(* CODESYS project CtaAppBacNetKBOB_1.0.0.0.library
   Description: CtaAppBacNetKBOB Library der CTA
   Version: 1.0.0.0
   Title: CtaAppBacNetKBOB
   Author: SIS
   Company: CTA
   DocFormat: reStructuredText
   Placeholder: CtaAppBacNetKBOB
   DefaultNamespace: CtaAppBacNetKBOB
   CompiledLibraryCompatibilityVersion: CODESYS V3.5 SP16 Patch 3
   LanguageModelAttribute: qualified-access-only

Project tree, tasks and I/O mapping:
  libraries: CtaAppBmk, 1.0.0.0 (CTA); Standard, 3.5.18.0 (System); CtaSysConfig, 1.0.0.0 (CTA); CmpDynamicText, 3.5.17.0 (System); WagoTypesBACnet, 1.0.9.7 (WAGO); SysProcess, 3.5.17.0 (System); CtaVisSymbols, 1.0.0.0 (CTA); StringUtils, 3.5.18.0 (System); SysTypes2 Interfaces, * (System); VisuSymbols, 4.5.0.0 (System); CtaVisHelp, 1.0.0.0 (CTA); WagoSysErrorBase, 1.6.2.6 (WAGO); WagoSysBACnet, 2.0.0.6 (WAGO); WagoSysVisuBACnet, 2.0.0.0 (WAGO)
  40 Visualizations/
    BACNET_PARAMETER/
      visualisation DIA_BACNET_PARAMETER
      visualisation VIS_DIA_BACNET_PARAMETER
      visualisation VIS_BACNET_APP
      visualisation DIA_BACNET_LIST
  30 Program Organization Units/
    FCs/
      XMLFcs/
        XMLBase/
          function fcXMLAddAttribute [ST]
          function fcXMLCheckNode [ST]
          function fcXMLDeleteNode [ST]
          function fcXMLUpdateAttribute [ST]
          function fcXMLUpdateNode [ST]
          function fcXMLAddNode [ST]
        XML BacNet Override/
          DELETENODE/
            function fcXMLDeleteOverrideNode [ST]
          STRUCTUREDVIEW/
            function fcXMLStructuredView [ST]
            function fcXMLAddStructuredViewToDevice [ST]
            function fcXMLDeleteStructuredViewFromDevice [ST]
          TRENDLOG/
            function fcXMLTrendLogOverride [ST]
          DEVICE/
            function fcXMLDeviceOverride [ST]
      BacNetId/
        function fcDWordToHexString [ST]
        function fcBacNetIdToIdWitType [ST]
      BmkToAdr/
        function fcBmkToAdr [ST]
      BacNetText/
        function fcGetBcText [ST]
      UTF8Fcs/
        function fcAsciiToUtf [ST]
        function fcUtfToAscii [ST]
      BacNetIni/
        function fcBacNetIni [ST]
    FBs/
      AT_FUNKTIONEN/
        AT_MESSWERTGEBER_BINÄR/
          function block FB_AT_MESSWERTGEBER_BINÄR [ST]: metDELETE, metCREATE, metCreate_A_BI_1, metCreate_B_TL_1, metCreate_C_BV_1, metCREATE_KBOB_2017_V1, metCREATE_STRUCTVIEW_KBOB_2017_V1, metCREATE_STRUCTVIEW_KBOB_2021_V2, metCREATE_KBOB_2021_V2, FB_EXIT, metCYCLIC_DESCRIPTION_FIX, metCYCLIC_KBOB_2017_V1, metCYCLIC_KBOB_2021_V2
        AT_MESSWERTGEBER_STETIG/
          function block FB_AT_MESSWERTGEBER_STETIG [ST]: metDELETE, FB_EXIT, metCREATE, metCreate_A_AI_1, metCreate_C_TL_1, metCreate_B_EE_1, metCREATE_KBOB_2017_V1, metCREATE_STRUCTVIEW_KBOB_2017_V1, metCREATE_KBOB_2021_V2, metCREATE_STRUCTVIEW_KBOB_2021_V2, metCYCLIC_KBOB_2017_V1, metCYCLIC_KBOB_2021_V2, metCYCLIC_DESCRIPTION_FIX
        AT_ANTRIEB_STETIG/
          function block FB_AT_ANTRIEB_STETIG [ST]: metCYCLIC_KBOB_2017_V1, metCYCLIC_KBOB_2021_V2, metCYCLIC_DESCRIPTION_FIX, FB_EXIT, metDELETE, metCREATE_KBOB_2017_V1, metCREATE_STRUCTVIEW_KBOB_2017_V1, metCREATE_STRUCTVIEW_KBOB_2021_V2, metCREATE_KBOB_2021_V2, metCREATE, metCreate_F_BI_1, metCreate_G_AO_1, metCreate_I_AI_1, metCreate_K_BI_2, metCreate_L_BV_3, metCreate_H_TL_2, metCreate_J_TL_3, metCreate_A_BO_1, metCreate_B_TL_1, metCreate_C_EE_1, metCreate_E_BV_2
        AT_ANLAGENSCHALTER/
          function block FB_AT_ANLAGENSCHALTER [ST]: FB_EXIT, metCREATE, metCreate_A_MV_1, metCreate_B_MI_1, metCreate_C_BV_1, metCreate_D_SC_1, metCREATE_KBOB_2017_V1, metCREATE_STRUCTVIEW_KBOB_2017_V1, metCREATE_KBOB_2021_V2, metCREATE_STRUCTVIEW_KBOB_2021_V2, metDELETE, metCYCLIC_KBOB_2017_V1, metCYCLIC_KBOB_2021_V2, metCYCLIC_DESCRIPTION_FIX
        AT_AUTOMATIONSTATION/
          function block FB_AT_AUTOMATIONSSTATION [ST]: metCYCLIC_KBOB_2017_V1, metCYCLIC_KBOB_2021_V2, metCYCLIC_DESCRIPTION_FIX, FB_EXIT, metDELETE, metCREATE_KBOB_2017_V1, metCREATE_STRUCTVIEW_KBOB_2017_V1, metCREATE_KBOB_2021_V2, metCREATE_STRUCTVIEW_KBOB_2021_V2, metCREATE, metCreate_L_NC_160, metCreate_L_NC_161, metCreate_L_NC_162, metCreate_L_NC_163, metCreate_M_NC_192, metCreate_M_NC_193, metCreate_N_NC_224, metCreate_N_NC_225, metCreate_O_BV_1, metCreate_P_BV_2, metCreate_Q_BV_3, metCreate_R_BV_4, metCreate_S_BV_5, metCreate_I_NC_66, metCreate_J_NC_97, metCreate_J_NC_98, metCreate_J_NC_99, metCreate_K_NC_128, metCreate_H_NC_35, metCreate_I_NC_64, metCreate_I_NC_67, metCreate_J_NC_96, metCreate_K_NC_129, metCreate_K_NC_130, metCreate_K_NC_131, metCreate_A_DV_1, metCreate_B_CL_1, metCreate_C_CL_2, metCreate_D_CL_3, metCreate_E_CL_4, metCreate_F_EL_1, metCreate_G_NC_1, metCreate_G_NC_2, metCreate_G_NC_3, metCreate_G_NC_4, metCreate_H_NC_32, metCreate_H_NC_33, metCreate_H_NC_34, metCreate_I_NC_65
        AT_ANLAGEFUNKTION/
          function block FB_AT_ANLAGEFUNKTION [ST]: metCREATE_STRUCTVIEW_KBOB_2021_V2, metCREATE_KBOB_2021_V2, metCreate_H_BO_2, metCreate_I_BO_3, metCreate_D_BV_4, metCreate_E_BI_1, metCreate_B_BV_2, metCreate_C_BV_3, metCreate_J_SC_1, metCreate_F_BV_5, metCreate_G_BO_1, metCreate_A_BV_1, metCREATE_KBOB_2017_V1, metCREATE_STRUCTVIEW_KBOB_2017_V1, metCREATE, metCYCLIC_KBOB_2017_V1, metCYCLIC_KBOB_2021_V2, metCYCLIC_DESCRIPTION_FIX, FB_EXIT, metDELETE
        AT_ZÄHLER/
          function block FB_AT_ZÄHLER [ST]: metCREATE_STRUCTVIEW_KBOB_2021_V2, metCREATE_KBOB_2021_V2, metCreate_A_AV_1, metCreate_B_TL_1, metCreate_C_BV_1, metCREATE, metCREATE_KBOB_2017_V1, metCREATE_STRUCTVIEW_KBOB_2017_V1, metDELETE, FB_EXIT, metCYCLIC_DESCRIPTION_FIX, metCYCLIC_KBOB_2017_V1, metCYCLIC_KBOB_2021_V2
        AT_STELLORGAN_STETIG/
          function block FB_AT_AT_STELLORGAN_STETIG [ST]: metCREATE_STRUCTVIEW_KBOB_2021_V2, metCREATE_KBOB_2021_V2, metCreate_D_BI_1, metCreate_A_AO_1, metCreate_C_TL_1, metCreate_E_BI_2, metCreate_B_AI_1, metCreate_F_BV_1, metCREATE_KBOB_2017_V1, metCREATE_STRUCTVIEW_KBOB_2017_V1, metCREATE, metCYCLIC_KBOB_2017_V1, metCYCLIC_KBOB_2021_V2, metCYCLIC_DESCRIPTION_FIX, FB_EXIT, metDELETE
      BACNET_PARAMETER/
        function block FB_BACNET_PARAMETER [ST]: proCreate, proDelete, proUseAKS, proInitDone, CONFIG, metRequestDelete, metGetTextListName, proKBOB_REV, P_fbenBacNetKbobRev, P_fbxEnableBacNet, P_fbxUseAKS, P_fbxUseExklTxtList, proTimeToOnline, proDestroyBacNetOverrideXmlNode, proRebootRequired, metAddObj, BACNETLIBPARACHECK, P_fbdiDeviceId, P_fbxAnsiCodiert
      OBJ_IDENTIFER_BASE/
        function block FB_OBJ_ID_BASE [ST]: OBJ_ID_BASE, OBJ_NAME_BASE, OBJ_NAME_DESCRIPTION, metCREATE, metDELETE, FB_EXIT, FB_INIT, proINextObj, proIsCreatet, proAllowCreate, proAllowDelete
    Pou/
      program BAC_NET [ST]
  00000000-0000-0000-0000-000000000000|D:\CoDeSys\LibrariesV3\trunk\Intern\CAA\CAA Template\3.4.0.0 draft\Placeholder.xml
  00000000-0000-0000-0000-000000000000|D:\CoDeSys\LibrariesV3\trunk\Intern\CAA\CAA Template\3.2.0.3 draft\Prefix.pdf
  00000000-0000-0000-0000-000000000000|D:\CoDeSys\LibrariesV3\trunk\Intern\CAA\CAA Template\3.5.2.0 draft\Placeholder.xml
  20 Structs/
    ENUMERATION/
      data type enTypeOfBacNetFunktion
      data type enEvent
      data type enTypeOfBacNetTextList
      data type enKBOB_REV
  50 Images/
  10 Documenation/
    global variables VersionHistory
    global variables readMe
  21 Interface/
    BACNET_PARAMETER/
      interface ITF_BACNET_PARAMETER: metGetTextListName, metRequestDelete, proCreate, proDelete, proInitDone, proKBOB_REV, proUseAKS, P_fbxEnableBacNet, P_fbxUseAKS, P_fbxUseExklTxtList, P_fbenBacNetKbobRev, proTimeToOnline, metAddObj, proRebootRequired, proDestroyBacNetOverrideXmlNode, P_fbdiDeviceId, P_fbxAnsiCodiert
    OBJ_IDENTIFER_BASE/
      interface ITF_OBJ_ID_BASE: FB_EXIT, metCREATE, OBJ_ID_BASE, OBJ_NAME_BASE, OBJ_NAME_DESCRIPTION, metDELETE, proINextObj, proAllowCreate, proIsCreatet, proAllowDelete
  11 Library Parameter/
  12 Konstanten/
  60 Textlisten/
    AT_FUNKTIONEN_TEXTLISTEN/
      AT_ANLAGENSCHALTER/
        text list TXT_AT_ANLAGENSCHALTER_NC
        text list TXT_AT_ANLAGENSCHALTER_ENDING
        text list TXT_AT_ANLAGENSCHALTER_EVENTMESSAGE
        text list TXT_AT_ANLAGENSCHALTER_PRESV
        text list TXT_AT_ANLAGENSCHALTER_DESCRIPTION
      AT_ANTRIEB_STETIG/
        text list TXT_AT_ANTRIEB_STETIG_ENDING
        text list TXT_AT_ANTRIEB_STETIG_DESCRIPTION
        text list TXT_AT_ANTRIEB_STETIG_PRESV
        text list TXT_AT_ANTRIEB_STETIG_EVENTMESSAGE
        text list TXT_AT_ANTRIEB_STETIG_NC
      AT_MESSWERTGEBER_BINÄR/
        text list TXT_AT_MESSWERTGEBER_BINAR_DESCRIPTION
        text list TXT_AT_MESSWERTGEBER_BINAR_ENDING
        text list TXT_AT_MESSWERTGEBER_BINAR_NC
        text list TXT_AT_MESSWERTGEBER_BINAR_EVENTMESSAGE
        text list TXT_AT_MESSWERTGEBER_BINAR_PRESV
      AT_MESSWERTGEBER_STETIG/
        text list TXT_AT_MESSWERTGEBER_STETIG_NC
        text list TXT_AT_MESSWERTGEBER_STETIG_DESCRIPTION
        text list TXT_AT_MESSWERTGEBER_STETIG_ENDING
        text list TXT_AT_MESSWERTGEBER_STETIG_EVENTMESSAGE
        text list TXT_AT_MESSWERTGEBER_STETIG_PRESV
      AT_AUTOMATIONSTATION/
        text list TXT_AT_AUTOMATIONSSTATION_DESCRIPTION
        text list TXT_AT_AUTOMATIONSSTATION_ENDING
        text list TXT_AT_AUTOMATIONSSTATION_NC
        text list TXT_AT_AUTOMATIONSSTATION_PRESV
        text list TXT_AT_AUTOMATIONSSTATION_EVENTMESSAGE
      AT_ANLAGEFUNKTION/
        text list TXT_AT_ANLAGEFUNKTION_DESCRIPTION
        text list TXT_AT_ANLAGEFUNKTION_ENDING
        text list TXT_AT_ANLAGEFUNKTION_EVENTMESSAGE
        text list TXT_AT_ANLAGEFUNKTION_NC
        text list TXT_AT_ANLAGEFUNKTION_PRESV
      AT_ZÄHLER/
        text list TXT_AT_ZÄHLER_DESCRIPTION
        text list TXT_AT_ZÄHLER_ENDING
        text list TXT_AT_ZÄHLER_EVENTMESSAGE
        text list TXT_AT_ZÄHLER_NC
        text list TXT_AT_ZÄHLER_PRESV
      AT_STELLORGAN_STETIG/
        text list TXT_AT_STELLORGAN_STETIG_ENDING
        text list TXT_AT_STELLORGAN_STETIG_EVENTMESSAGE
        text list TXT_AT_STELLORGAN_STETIG_DESCRIPTION
        text list TXT_AT_STELLORGAN_STETIG_NC
        text list TXT_AT_STELLORGAN_STETIG_PRESV
    KBOB/
      text list KBOB_REV_TXT
  13 Globale Variablen/
    global variables GVL_BACNET
  text list GlobalTextList
*)

// 20 Structs/ENUMERATION/enTypeOfBacNetFunktion
{attribute 'qualified_only'}
TYPE enTypeOfBacNetFunktion :
(
	Type_Anlagenschalter            := 01,
    Type_AntriebStetig              := 02,
    Type_AbsperrStellorgan2p        := 03,
    Type_AbsperrStellorganStetig    := 04,
    Type_MesswertgeberStetig        := 05,
    Type_MesswertgeberBinär         := 06,
    Type_ParameterAnalog            := 07,
    Type_ParameterBinär             := 08,
	Type_Automationsstation			:= 09,
	Type_Anlagefunktion				:= 10,
	Type_Zähler						:= 11
);
END_TYPE

// 20 Structs/ENUMERATION/enEvent
{attribute 'qualified_only'}
{attribute 'strict'}
TYPE enEvent :
(
	ToOffNormal := 1,
	ToFault		:= 2,
	ToNormal	:= 3
);
END_TYPE

// 20 Structs/ENUMERATION/enTypeOfBacNetTextList
{attribute 'qualified_only'}
{attribute 'strict'}
TYPE enTypeOfBacNetTextList :
(
	ENDING 			:= 0,
	DESCRIPTION		:= 1,
	NC				:= 2,
	EVENTMESSAGE	:= 3,
	PRESENTVALUE	:= 4
);
END_TYPE

// 20 Structs/ENUMERATION/enKBOB_REV
{attribute 'qualified_only'}
TYPE enKBOB_REV :
(
	
	KBOB_REV2017_V1 := 0,
	KBOB_REV2021_V2 := 1
);
END_TYPE

// 10 Documenation/VersionHistory
(* 

.. image:: ../../Images/CTA_Logo.jpg
   :align: right
   :width: 15% 

**Vorlage**   


============ =========== =========== ============================================
**Date**     **Version** **Author**  **Change**
------------ ----------- ----------- --------------------------------------------
04.03.2021   0.0.0.0     SIS         Vorlage erstellt

============ =========== =========== ============================================


*)
VAR_GLOBAL
    stInfo : STRING:= '0.0.0.0, Vorlage, CTA';
END_VAR

// 10 Documenation/readMe
(*

**ReadMe**
 
|	**Empfehlung**
|
|	Dokumentrieren Sie die Library für eine nachhaltige Entwicklung
|     
| *Beispiel* 
|
| Dies ist die Vorlage Library der CTA. Erstellen Sie ihre Library anhand dieser Vorlage.
*)

VAR_GLOBAL
    xReadMeDone              :   BOOL;
END_VAR

// 13 Globale Variablen/GVL_BACNET
{attribute 'qualified_only'}
{attribute 'global_init_slot' := '49989'}
VAR_GLOBAL
	fbBacNetBmkDevice			:	CtaAppBmk.fbBMK := (stObjId := 'BacNetDevice');
	fbBacNetParameter			:	FB_BACNET_PARAMETER;
	fbAtAutomationsstation		:	FB_AT_AUTOMATIONSSTATION := (ITF_BMK_IN := fbBacNetBmkDevice);
	stBacNetDeviceId			:	STRING(8);
END_VAR

// 30 Program Organization Units/FCs/XMLFcs/XMLBase/fcXMLAddAttribute
FUNCTION fcXMLAddAttribute : BOOL
VAR_INPUT
	stParentPath			:	STRING(100);	// Start with '//*/
	stNodeName				:	STRING(100);
	stAttribute1			:	STRING(100);
	stAttribute1Value		:	STRING(150);
	stAttribute2Check		:	STRING(100);
	stAttribute2ValueCheck	:	STRING(150);
	stXmlFilePathName		:	STRING(255);
	xIgnoreCheck			:	BOOL;
END_VAR
VAR
	stCommand			:	STRING(1000);
	stTemp				:	STRING(255);
	stResult			:	STRING(255);
	RTS_IEC_RESULT		:	SysTypes.RTS_IEC_RESULT;
END_VAR

IF NOT fcXMLCheckNode(stParentPath,stNodeName,stAttribute1,stAttribute1Value,stAttribute2Check,stAttribute2ValueCheck,stXmlFilePathName) OR xIgnoreCheck THEN
	// create Attribute	
	stCommand := 	'';
	stTemp	  := 	'';
	stTemp	  :=	'xmlstarlet ed -L --insert "';
	StrConcatA(ADR(stTemp),ADR(stCommand),TO_INT(SIZEOF(stCommand)));
	stTemp	  := 	'';
	stTemp	  :=	stParentPath;
	StrConcatA(ADR(stTemp),ADR(stCommand),TO_INT(SIZEOF(stCommand)));
	stTemp	  := 	'';
	stTemp	  :=	'/';
	StrConcatA(ADR(stTemp),ADR(stCommand),TO_INT(SIZEOF(stCommand)));	
	stTemp	  := 	'';
	stTemp	  :=	stNodeName;
	StrConcatA(ADR(stTemp),ADR(stCommand),TO_INT(SIZEOF(stCommand)));	
	stTemp	  := 	'';
	stTemp	  :=	'[last()]" -t attr -n "';
	StrConcatA(ADR(stTemp),ADR(stCommand),TO_INT(SIZEOF(stCommand)));		
	stTemp	  := 	'';
	stTemp	  :=	stAttribute1;
	StrConcatA(ADR(stTemp),ADR(stCommand),TO_INT(SIZEOF(stCommand)));	
	stTemp	  := 	'';
	stTemp	  :=	'" -v "';
	StrConcatA(ADR(stTemp),ADR(stCommand),TO_INT(SIZEOF(stCommand)));	
	stTemp	  := 	'';
	stTemp	  :=	stAttribute1Value;
	StrConcatA(ADR(stTemp),ADR(stCommand),TO_INT(SIZEOF(stCommand)));
	stTemp	  := 	'';
	stTemp	  :=	'" ';
	StrConcatA(ADR(stTemp),ADR(stCommand),TO_INT(SIZEOF(stCommand)));
	stTemp	  := 	'';
	stTemp	  :=	stXmlFilePathName;
	StrConcatA(ADR(stTemp),ADR(stCommand),TO_INT(SIZEOF(stCommand)));	

	SysProcess_Implementation.SysProcessExecuteCommand(stCommand,ADR(RTS_IEC_RESULT));
	fcXMLAddAttribute := TRUE;
END_IF;

END_FUNCTION

// 30 Program Organization Units/FCs/XMLFcs/XMLBase/fcXMLCheckNode
FUNCTION fcXMLCheckNode : BOOL
VAR_INPUT
	stParentPath			:	STRING(100);	// Start with '//*/
	stNodeName				:	STRING(100);
	stAttribute1			:	STRING(100);
	stAttribute1Value		:	STRING(150);
	stAttribute2			:	STRING(100);
	stAttribute2Value		:	STRING(150);
	stXmlFilePathName		:	STRING(255);
END_VAR
VAR
	stCommand			:	STRING(1000);
	stTemp				:	STRING(255);
	stResult			:	STRING(255);
	RTS_IEC_RESULT		:	SysTypes.RTS_IEC_RESULT;
END_VAR

stCommand := 	'';
stTemp	  := 	'';
stTemp	  :=	'xmlstarlet sel -t -v "count(';
StrConcatA(ADR(stTemp),ADR(stCommand),TO_INT(SIZEOF(stCommand)));
stTemp	  := 	'';
stTemp	  :=	stParentPath;
StrConcatA(ADR(stTemp),ADR(stCommand),TO_INT(SIZEOF(stCommand)));
stTemp	  := 	'';
stTemp	  :=	'/';
StrConcatA(ADR(stTemp),ADR(stCommand),TO_INT(SIZEOF(stCommand)));
stTemp	  := 	'';
stTemp	  :=	stNodeName;
StrConcatA(ADR(stTemp),ADR(stCommand),TO_INT(SIZEOF(stCommand)));
stTemp	  := 	'';
stTemp	  :=	SEL(stAttribute1 <> '',' ','[@');
StrConcatA(ADR(stTemp),ADR(stCommand),TO_INT(SIZEOF(stCommand)));
stTemp	  := 	'';
stTemp	  :=	stAttribute1;
StrConcatA(ADR(stTemp),ADR(stCommand),TO_INT(SIZEOF(stCommand)));
stTemp	  := 	'';
stTemp	  :=	SEL(stAttribute1 <> '',' ','=$'');
StrConcatA(ADR(stTemp),ADR(stCommand),TO_INT(SIZEOF(stCommand)));
stTemp	  := 	'';
stTemp	  :=	SEL(stAttribute1 <> '','',stAttribute1Value);
StrConcatA(ADR(stTemp),ADR(stCommand),TO_INT(SIZEOF(stCommand)));
stTemp	  := 	'';
stTemp	  :=	SEL(stAttribute1 <> '','',SEL(stAttribute2 <> '','$']','$' and @'));
StrConcatA(ADR(stTemp),ADR(stCommand),TO_INT(SIZEOF(stCommand)));
stTemp	  := 	'';
stTemp	  :=	stAttribute2;
StrConcatA(ADR(stTemp),ADR(stCommand),TO_INT(SIZEOF(stCommand)));
stTemp	  := 	'';
stTemp	  :=	SEL(stAttribute2 <> '',' ','=$'');
StrConcatA(ADR(stTemp),ADR(stCommand),TO_INT(SIZEOF(stCommand)));
stTemp	  := 	'';
stTemp	  :=	SEL(stAttribute2 <> '','',stAttribute2Value);
StrConcatA(ADR(stTemp),ADR(stCommand),TO_INT(SIZEOF(stCommand)));
stTemp	  := 	'';
stTemp	  :=	SEL(stAttribute2 <> '','','$']');
StrConcatA(ADR(stTemp),ADR(stCommand),TO_INT(SIZEOF(stCommand)));
stTemp	  := 	'';
stTemp	  :=	')" ';
StrConcatA(ADR(stTemp),ADR(stCommand),TO_INT(SIZEOF(stCommand)));
stTemp	  := 	'';
stTemp	  :=	stXmlFilePathName;
StrConcatA(ADR(stTemp),ADR(stCommand),TO_INT(SIZEOF(stCommand)));

SysProcess_Implementation.SysProcessExecuteCommand2(stCommand,stResult,SIZEOF(stResult),ADR(RTS_IEC_RESULT));

IF stResult ='0' OR stResult ='' THEN
	fcXMLCheckNode := FALSE;
ELSE
	fcXMLCheckNode := TRUE;
END_IF

END_FUNCTION

// 30 Program Organization Units/FBs/AT_FUNKTIONEN/AT_MESSWERTGEBER_BINÄR/FB_AT_MESSWERTGEBER_BINÄR
FUNCTION_BLOCK FB_AT_MESSWERTGEBER_BINÄR EXTENDS FB_OBJ_ID_BASE
VAR_INPUT
	xValue				:	BOOL;
	xError				:	BOOL;
END_VAR
VAR_OUTPUT

END_VAR
VAR
	(* BacNet Objects *)
	A_BI_1		:	WagoSysBACnet.FbBinaryInput_large(-1);					// Istwert
	B_TL_1		:	WagoSysBACnet.FbTrendLog_large(-1);                     // Aufzeichnung Istwert
	C_BV_1		:	WagoSysBACnet.FbBinaryValue_large(-1);              	// Störung

END_VAR
VAR CONSTANT
	usiAnzBacNetObj	:	USINT	:= 3;
END_VAR

(* Call Base FB*)
SUPER^();
(* Cyclic Action *)
IF xCreatet THEN
	(* DESCTIPTION FIX *)
	metCYCLIC_DESCRIPTION_FIX();
	(* Get Revision *)
	CASE GVL_BACNET.fbBacNetParameter.proKBOB_REV OF
		(* KBOB 2021 V2 *)
		enKBOB_REV.KBOB_REV2021_V2:
			metCYCLIC_KBOB_2021_V2();
		(* KBOB 2017 V1 *)
		enKBOB_REV.KBOB_REV2017_V1:
			metCYCLIC_KBOB_2017_V1();
		(* Default *)
		ELSE
			metCYCLIC_KBOB_2021_V2();
	END_CASE;	
END_IF;

METHOD metDELETE : BOOL
VAR_INPUT
END_VAR
VAR
	oStatus		:	WagoSysErrorBase.FbResult;
	usiErrors	:	USINT;
END_VAR
(* A_BO_1*)
IF A_BI_1.xIsCreated THEN
	A_BI_1.Delete(oStatus=>oStatus);	
END_IF;
(* B_TL_1 *)
IF B_TL_1.xIsCreated THEN
	IF GVL_BACNET.fbBacNetParameter.proDestroyBacNetOverrideXmlNode THEN
		fcXMLDeleteOverrideNode(fcBacNetIdToIdWitType(B_TL_1.IObjectIdentifier.diInstance,B_TL_1.IObjectIdentifier.eObjectType));
	END_IF;
	B_TL_1.Delete(oStatus=>oStatus);
END_IF;
(* C_BV_1 *)
IF C_BV_1.xIsCreated THEN
	C_BV_1.Delete(oStatus=>oStatus);
END_IF;
(* Delete Struct View *)
IF GVL_BACNET.fbBacNetParameter.proDestroyBacNetOverrideXmlNode THEN
	fcXMLDeleteOverrideNode(fcBacNetIdToIdWitType(TO_DINT(CONCAT(TO_STRING(OBJ_ID_BASE),'1')),WagoTypesBacNet.eBACnetObjectType.BACnet_structured_view));
	fcXMLDeleteStructuredViewFromDevice(fcBacNetIdToIdWitType(TO_DINT(CONCAT(TO_STRING(OBJ_ID_BASE),'1')),WagoTypesBacNet.eBACnetObjectType.BACnet_structured_view));
END_IF;
metDELETE :=	A_BI_1.xIsCreated OR
				B_TL_1.xIsCreated OR
				C_BV_1.xIsCreated;
(* Reset Create Case *)
usiCreateCase := 1;
END_METHOD

METHOD metCREATE : BOOL;
VAR_INPUT
END_VAR
VAR
	usiErrors	:	USINT;
END_VAR
(* Get Revision *)
CASE GVL_BACNET.fbBacNetParameter.proKBOB_REV OF
	(* KBOB 2021 V2 *)
	enKBOB_REV.KBOB_REV2021_V2:
		usiErrors := usiErrors + TO_USINT(NOT metCREATE_KBOB_2021_V2());
	(* KBOB 2017 V1 *)
	enKBOB_REV.KBOB_REV2017_V1:
		usiErrors := usiErrors + TO_USINT(NOT metCREATE_KBOB_2017_V1());
	(* Default *)
	ELSE
		usiErrors := usiErrors + TO_USINT(NOT metCREATE_KBOB_2021_V2());
END_CASE;

(* OK = 0*)
xErrorCreate := TO_BOOL(usiErrors);
metCREATE := NOT TO_BOOL(usiErrors) AND usiCreateCase = usiAnzBacNetObj;
END_METHOD

METHOD metCreate_A_BI_1 : BOOL
(* A_BI_1*)
IF NOT A_BI_1.xIsCreated THEN
	(* Ziel						UTF8->ASCII						OBJ_NAME_BASE			BacNet Text		Textlistname									BacNet Funktion																	BacNet Textlist type												TextId		*)
	A_BI_1._sObjectName		:=	fcUtfToAscii(Standard.CONCAT(	OBJ_NAME_BASE		,	fcGetBcText(	GVL_BACNET.fbBacNetParameter.metGetTextListName(enTypeOfBacNetFunktionIn := enTypeOfBacNetFunktion.Type_MesswertgeberBinär,		enTypeOfBacNetTextListIn := enTypeOfBacNetTextList.ENDING		),	'A_BI_1')));
	A_BI_1._sDescription	:= 	fcUtfToAscii(Standard.CONCAT(	OBJ_NAME_DESCRIPTION,	fcGetBcText(	GVL_BACNET.fbBacNetParameter.metGetTextListName(enTypeOfBacNetFunktionIn := enTypeOfBacNetFunktion.Type_MesswertgeberBinär,		enTypeOfBacNetTextListIn := enTypeOfBacNetTextList.DESCRIPTION	),	'A_BI_1')));
	(* Create Id from Base Id and Object Nr (Last nummber of Name *)	
	A_BI_1.Create(diInstance := TO_DINT(Standard.CONCAT(TO_STRING(dwOBJ_ID_BASE),'1')));
	(* Check if Created *)
	IF A_BI_1.xIsCreated THEN
		(* Set Group *)
		A_BI_1.setPropertyGroup(WagoTypesBacNet.eBACnetPropertyIdentifier.PROP_PRESENT_VALUE						,WagoTypesBacNet.eBACnetPropertyUpdateGroup.GROUP_CYCLIC);
		A_BI_1.setPropertyGroup(WagoTypesBacNet.eBACnetPropertyIdentifier.PROP_PRIORITY_ARRAY						,WagoTypesBacNet.eBACnetPropertyUpdateGroup.GROUP_CYCLIC);
		A_BI_1.setPropertyGroup(WagoTypesBacNet.eBACnetPropertyIdentifier.PROP_ELAPSED_ACTIVE_TIME					,WagoTypesBacNet.eBACnetPropertyUpdateGroup.GROUP_CYCLIC);
		A_BI_1.setPropertyGroup(WagoTypesBacNet.eBACnetPropertyIdentifier.PROP_DESCRIPTION							,WagoTypesBacNet.eBACnetPropertyUpdateGroup.GROUP_CYCLIC);
		A_BI_1.setPropertyGroup(WagoTypesBacNet.eBACnetPropertyIdentifier.PROP_EVENT_MESSAGE_TEXTS_CONFIG			,WagoTypesBacNet.eBACnetPropertyUpdateGroup.GROUP_CYCLIC);
		(* Set Description to Overwrite retain*)
		A_BI_1.sDescription	:= A_BI_1._sDescription;
		(* Ziel												UTF8->ASCII		BacNet Text		Textlistname									BacNet Funktion																	BacNet Textlist type												TextId		*)
		A_BI_1.IEventMessageTextsConfig.sToOffNormal	:=	fcUtfToAscii(	fcGetBcText(	GVL_BACNET.fbBacNetParameter.metGetTextListName(enTypeOfBacNetFunktionIn := enTypeOfBacNetFunktion.Type_MesswertgeberBinär,		enTypeOfBacNetTextListIn := enTypeOfBacNetTextList.EVENTMESSAGE	),	'A_BI_1_ToOffNormal'	));		
		A_BI_1.IEventMessageTextsConfig.sToFault		:=	fcUtfToAscii(	fcGetBcText(	GVL_BACNET.fbBacNetParameter.metGetTextListName(enTypeOfBacNetFunktionIn := enTypeOfBacNetFunktion.Type_MesswertgeberBinär,		enTypeOfBacNetTextListIn := enTypeOfBacNetTextList.EVENTMESSAGE	),	'A_BI_1_ToFault'		));		
		A_BI_1.IEventMessageTextsConfig.sToNormal		:=	fcUtfToAscii(	fcGetBcText(	GVL_BACNET.fbBacNetParameter.metGetTextListName(enTypeOfBacNetFunktionIn := enTypeOfBacNetFunktion.Type_MesswertgeberBinär,		enTypeOfBacNetTextListIn := enTypeOfBacNetTextList.EVENTMESSAGE	),	'A_BI_1_ToNormal'		));		

		(* Ziel												UTF8->ASCII		BacNet Text		Textlistname									BacNet Funktion																	BacNet Textlist type												TextId		*)	
		A_BI_1.sActiveText								:= 	fcUtfToAscii(	fcGetBcText(	GVL_BACNET.fbBacNetParameter.metGetTextListName(enTypeOfBacNetFunktionIn := enTypeOfBacNetFunktion.Type_MesswertgeberBinär,		enTypeOfBacNetTextListIn := enTypeOfBacNetTextList.PRESENTVALUE	),	'A_BI_1_ST_ACTIVE'		));
		A_BI_1.sInactiveText							:= 	fcUtfToAscii(	fcGetBcText(	GVL_BACNET.fbBacNetParameter.metGetTextListName(enTypeOfBacNetFunktionIn := enTypeOfBacNetFunktion.Type_MesswertgeberBinär,		enTypeOfBacNetTextListIn := enTypeOfBacNetTextList.PRESENTVALUE	),	'A_BI_1_ST_INACTIVE'	));	

		(* Ziel												Convert			BacNet Text		Textlistname									BacNet Funktion																	BacNet Textlist type												TextId		*)	
		A_BI_1.udiNotificationClass						:= 	TO_UDINT	(	fcGetBcText(	GVL_BACNET.fbBacNetParameter.metGetTextListName(enTypeOfBacNetFunktionIn := enTypeOfBacNetFunktion.Type_MesswertgeberBinär,		enTypeOfBacNetTextListIn := enTypeOfBacNetTextList.NC			),	'A_BI_1_NC'	));	
		A_BI_1.eNotifyType								:= 	WagoTypesBACnet.eBACnetNotifyType.NOTIFY_TYPE_EVENT;
		A_BI_1.xAlarmValue								:= 	TO_BOOL		(	fcGetBcText(	GVL_BACNET.fbBacNetParameter.metGetTextListName(enTypeOfBacNetFunktionIn := enTypeOfBacNetFunktion.Type_MesswertgeberBinär,		enTypeOfBacNetTextListIn := enTypeOfBacNetTextList.NC			),	'A_BI_1_ALV'	));	
		
	ELSE
		A_BI_1.Delete();
	END_IF;
	(* Get Status *)
	metCreate_A_BI_1 := A_BI_1.xIsCreated;	
END_IF;
END_METHOD

METHOD metCreate_B_TL_1 : BOOL
(* B_TL_1*)
IF NOT B_TL_1.xIsCreated THEN
	(* Ziel						UTF8->ASCII						OBJ_NAME_BASE			BacNet Text		Textlistname									BacNet Funktion																BacNet Textlist type												TextId		*)
	B_TL_1._sObjectName		:=	fcUtfToAscii(Standard.CONCAT(	OBJ_NAME_BASE		,	fcGetBcText(	GVL_BACNET.fbBacNetParameter.metGetTextListName(enTypeOfBacNetFunktionIn := enTypeOfBacNetFunktion.Type_MesswertgeberBinär,		enTypeOfBacNetTextListIn := enTypeOfBacNetTextList.ENDING		),	'B_TL_1')));
	B_TL_1._sDescription	:= 	fcUtfToAscii(Standard.CONCAT(	OBJ_NAME_DESCRIPTION,	fcGetBcText(	GVL_BACNET.fbBacNetParameter.metGetTextListName(enTypeOfBacNetFunktionIn := enTypeOfBacNetFunktion.Type_MesswertgeberBinär,		enTypeOfBacNetTextListIn := enTypeOfBacNetTextList.DESCRIPTION	),	'B_TL_1')));
	(* Create Id from Base Id and Object Nr (Last nummber of Name *)	
	B_TL_1.Create(diInstance := TO_DINT(Standard.CONCAT(TO_STRING(dwOBJ_ID_BASE),'1')));
	(* Check if Created *)
	IF B_TL_1.xIsCreated THEN
		(* Set Group *)
		B_TL_1.setPropertyGroup(WagoTypesBacNet.eBACnetPropertyIdentifier.PROP_PRESENT_VALUE						,WagoTypesBacNet.eBACnetPropertyUpdateGroup.GROUP_CYCLIC);
		B_TL_1.setPropertyGroup(WagoTypesBacNet.eBACnetPropertyIdentifier.PROP_PRIORITY_ARRAY						,WagoTypesBacNet.eBACnetPropertyUpdateGroup.GROUP_CYCLIC);
		B_TL_1.setPropertyGroup(WagoTypesBacNet.eBACnetPropertyIdentifier.PROP_ELAPSED_ACTIVE_TIME					,WagoTypesBacNet.eBACnetPropertyUpdateGroup.GROUP_CYCLIC);
		B_TL_1.setPropertyGroup(WagoTypesBacNet.eBACnetPropertyIdentifier.PROP_DESCRIPTION							,WagoTypesBacNet.eBACnetPropertyUpdateGroup.GROUP_CYCLIC);
		B_TL_1.setPropertyGroup(WagoTypesBacNet.eBACnetPropertyIdentifier.PROP_EVENT_MESSAGE_TEXTS_CONFIG			,WagoTypesBacNet.eBACnetPropertyUpdateGroup.GROUP_CYCLIC);
		(* Crate Override *)
		fcXMLTrendLogOverride(B_TL_1,A_BI_1.IObjectIdentifier,WagoTypesBacNet.eBACnetPropertyIdentifier.PROP_PRESENT_VALUE);
		(* Set Description to Overwrite retain*)
		B_TL_1.sDescription	:= B_TL_1._sDescription;
		(* Ziel												UTF8->ASCII		BacNet Text		Textlistname									BacNet Funktion																BacNet Textlist type												TextId		*)
		B_TL_1.IEventMessageTextsConfig.sToOffNormal	:=	fcUtfToAscii(	fcGetBcText(	GVL_BACNET.fbBacNetParameter.metGetTextListName(enTypeOfBacNetFunktionIn := enTypeOfBacNetFunktion.Type_MesswertgeberBinär,		enTypeOfBacNetTextListIn := enTypeOfBacNetTextList.EVENTMESSAGE	),	'B_TL_1_ToOffNormal'	));		
		B_TL_1.IEventMessageTextsConfig.sToFault		:=	fcUtfToAscii(	fcGetBcText(	GVL_BACNET.fbBacNetParameter.metGetTextListName(enTypeOfBacNetFunktionIn := enTypeOfBacNetFunktion.Type_MesswertgeberBinär,		enTypeOfBacNetTextListIn := enTypeOfBacNetTextList.EVENTMESSAGE	),	'B_TL_1_ToFault'		));		
		B_TL_1.IEventMessageTextsConfig.sToNormal		:=	fcUtfToAscii(	fcGetBcText(	GVL_BACNET.fbBacNetParameter.metGetTextListName(enTypeOfBacNetFunktionIn := enTypeOfBacNetFunktion.Type_MesswertgeberBinär,		enTypeOfBacNetTextListIn := enTypeOfBacNetTextList.EVENTMESSAGE	),	'B_TL_1_ToNormal'		));		

		(* Ziel												Convert			BacNet Text		Textlistname									BacNet Funktion																BacNet Textlist type												TextId		*)	
		B_TL_1.udiNotificationClass						:= 	TO_UDINT	(	fcGetBcText(	GVL_BACNET.fbBacNetParameter.metGetTextListName(enTypeOfBacNetFunktionIn := enTypeOfBacNetFunktion.Type_MesswertgeberBinär,		enTypeOfBacNetTextListIn := enTypeOfBacNetTextList.NC		),	'B_TL_1_NC'	));	
		B_TL_1.eNotifyType								:= 	WagoTypesBACnet.eBACnetNotifyType.NOTIFY_TYPE_EVENT;

		(* Logging Type *)
		B_TL_1.eLoggingType								:= WagoTypesBACnet.eBACnetLoggingType.LOGGING_TYPE_POLLED;
		
		(* Activate Logging *)
		B_TL_1.xEnable	:= TRUE;
	ELSE
		B_TL_1.Delete();
	END_IF;
	(* Get Status *)
	metCreate_B_TL_1 := B_TL_1.xIsCreated;	
END_IF;
END_METHOD

METHOD metCreate_C_BV_1 : BOOL
(* C_BV_1*)
IF NOT C_BV_1.xIsCreated THEN
	(* Ziel						UTF8->ASCII						OBJ_NAME_BASE			BacNet Text		Textlistname									BacNet Funktion																BacNet Textlist type												TextId		*)
	C_BV_1._sObjectName		:=	fcUtfToAscii(Standard.CONCAT(	OBJ_NAME_BASE		,	fcGetBcText(	GVL_BACNET.fbBacNetParameter.metGetTextListName(enTypeOfBacNetFunktionIn := enTypeOfBacNetFunktion.Type_MesswertgeberBinär,		enTypeOfBacNetTextListIn := enTypeOfBacNetTextList.ENDING		),	'C_BV_1')));
	C_BV_1._sDescription	:= 	fcUtfToAscii(Standard.CONCAT(	OBJ_NAME_DESCRIPTION,	fcGetBcText(	GVL_BACNET.fbBacNetParameter.metGetTextListName(enTypeOfBacNetFunktionIn := enTypeOfBacNetFunktion.Type_MesswertgeberBinär,		enTypeOfBacNetTextListIn := enTypeOfBacNetTextList.DESCRIPTION	),	'C_BV_1')));
	(* Create Id from Base Id and Object Nr (Last nummber of Name *)	
	C_BV_1.Create(diInstance := TO_DINT(Standard.CONCAT(TO_STRING(dwOBJ_ID_BASE),'1')));
	(* Check if Created *)
	IF C_BV_1.xIsCreated THEN
		(* Set Group *)
		C_BV_1.setPropertyGroup(WagoTypesBacNet.eBACnetPropertyIdentifier.PROP_PRESENT_VALUE						,WagoTypesBacNet.eBACnetPropertyUpdateGroup.GROUP_CYCLIC);
		C_BV_1.setPropertyGroup(WagoTypesBacNet.eBACnetPropertyIdentifier.PROP_PRIORITY_ARRAY						,WagoTypesBacNet.eBACnetPropertyUpdateGroup.GROUP_CYCLIC);
		C_BV_1.setPropertyGroup(WagoTypesBacNet.eBACnetPropertyIdentifier.PROP_ELAPSED_ACTIVE_TIME					,WagoTypesBacNet.eBACnetPropertyUpdateGroup.GROUP_CYCLIC);
		C_BV_1.setPropertyGroup(WagoTypesBacNet.eBACnetPropertyIdentifier.PROP_DESCRIPTION							,WagoTypesBacNet.eBACnetPropertyUpdateGroup.GROUP_CYCLIC);
		C_BV_1.setPropertyGroup(WagoTypesBacNet.eBACnetPropertyIdentifier.PROP_EVENT_MESSAGE_TEXTS_CONFIG			,WagoTypesBacNet.eBACnetPropertyUpdateGroup.GROUP_CYCLIC);
		(* Set Description to Overwrite retain*)
		C_BV_1.sDescription	:= C_BV_1._sDescription;
		(* Ziel												UTF8->ASCII		BacNet Text		Textlistname									BacNet Funktion																BacNet Textlist type												TextId		*)
		C_BV_1.IEventMessageTextsConfig.sToOffNormal	:=	fcUtfToAscii(	fcGetBcText(	GVL_BACNET.fbBacNetParameter.metGetTextListName(enTypeOfBacNetFunktionIn := enTypeOfBacNetFunktion.Type_MesswertgeberBinär,		enTypeOfBacNetTextListIn := enTypeOfBacNetTextList.EVENTMESSAGE	),	'C_BV_1_ToOffNormal'	));		
		C_BV_1.IEventMessageTextsConfig.sToFault		:=	fcUtfToAscii(	fcGetBcText(	GVL_BACNET.fbBacNetParameter.metGetTextListName(enTypeOfBacNetFunktionIn := enTypeOfBacNetFunktion.Type_MesswertgeberBinär,		enTypeOfBacNetTextListIn := enTypeOfBacNetTextList.EVENTMESSAGE	),	'C_BV_1_ToFault'		));		
		C_BV_1.IEventMessageTextsConfig.sToNormal		:=	fcUtfToAscii(	fcGetBcText(	GVL_BACNET.fbBacNetParameter.metGetTextListName(enTypeOfBacNetFunktionIn := enTypeOfBacNetFunktion.Type_MesswertgeberBinär,		enTypeOfBacNetTextListIn := enTypeOfBacNetTextList.EVENTMESSAGE	),	'C_BV_1_ToNormal'		));		

		(* Ziel												UTF8->ASCII		BacNet Text		Textlistname									BacNet Funktion																BacNet Textlist type												TextId		*)	
		C_BV_1.sActiveText								:= 	fcUtfToAscii(	fcGetBcText(	GVL_BACNET.fbBacNetParameter.metGetTextListName(enTypeOfBacNetFunktionIn := enTypeOfBacNetFunktion.Type_MesswertgeberBinär,		enTypeOfBacNetTextListIn := enTypeOfBacNetTextList.PRESENTVALUE	),	'C_BV_1_ST_ACTIVE'		));
		C_BV_1.sInactiveText							:= 	fcUtfToAscii(	fcGetBcText(	GVL_BACNET.fbBacNetParameter.metGetTextListName(enTypeOfBacNetFunktionIn := enTypeOfBacNetFunktion.Type_MesswertgeberBinär,		enTypeOfBacNetTextListIn := enTypeOfBacNetTextList.PRESENTVALUE	),	'C_BV_1_ST_INACTIVE'	));	

		(* Ziel												Convert			BacNet Text		Textlistname									BacNet Funktion																	BacNet Textlist type												TextId		*)	
		C_BV_1.udiNotificationClass						:= 	TO_UDINT	(	fcGetBcText(	GVL_BACNET.fbBacNetParameter.metGetTextListName(enTypeOfBacNetFunktionIn := enTypeOfBacNetFunktion.Type_MesswertgeberBinär,		enTypeOfBacNetTextListIn := enTypeOfBacNetTextList.NC			),	'C_BV_1_NC'	));	
		C_BV_1.eNotifyType								:= 	WagoTypesBACnet.eBACnetNotifyType.NOTIFY_TYPE_ALARM;		
		C_BV_1.xAlarmValue								:= 	TO_BOOL		(	fcGetBcText(	GVL_BACNET.fbBacNetParameter.metGetTextListName(enTypeOfBacNetFunktionIn := enTypeOfBacNetFunktion.Type_MesswertgeberBinär,		enTypeOfBacNetTextListIn := enTypeOfBacNetTextList.NC			),	'C_BV_1_ALV'	));	
		
	ELSE
		C_BV_1.Delete();
	END_IF;
	(* Get Status *)
	metCreate_C_BV_1 := C_BV_1.xIsCreated;	
END_IF;
END_METHOD

METHOD metCREATE_KBOB_2017_V1 : BOOL;
VAR_INPUT
END_VAR
VAR
	oStatus		:	WagoSysErrorBase.FbResult;
END_VAR
(* Resett *)
usiErrors := 0;	

(* Create Objeccts *)
CASE usiCreateCase OF
	1:	
		usiErrors := usiErrors + TO_USINT(NOT metCreate_A_BI_1());
	2:
		usiErrors := usiErrors + TO_USINT(NOT metCreate_B_TL_1());
	3:	
		usiErrors := usiErrors + TO_USINT(NOT metCreate_C_BV_1());
	0: 
		usiCreateCase := 1;
ELSE
	usiCreateCase := 0;
END_CASE;

(* STRUCT VIEW *)
metCREATE_STRUCTVIEW_KBOB_2017_V1();

(* OK = 0*)
metCREATE_KBOB_2017_V1 := NOT TO_BOOL(usiErrors);
END_METHOD

METHOD metCREATE_STRUCTVIEW_KBOB_2017_V1 : BOOL
VAR_INPUT
END_VAR
CASE usiCreateCase OF
	1:	
		fcXMLStructuredView(THIS^,A_BI_1.IObjectIdentifier);
	2:
		fcXMLStructuredView(THIS^,B_TL_1.IObjectIdentifier);
	3:
		fcXMLStructuredView(THIS^,C_BV_1.IObjectIdentifier);
		fcXMLAddStructuredViewToDevice(THIS^);
	0: 
		usiCreateCase := 1;
ELSE
	usiCreateCase := 0;
END_CASE
END_METHOD

METHOD metCREATE_STRUCTVIEW_KBOB_2021_V2 : BOOL
VAR_INPUT
END_VAR
CASE usiCreateCase OF
	1:	
		fcXMLStructuredView(THIS^,A_BI_1.IObjectIdentifier);
	2:
		fcXMLStructuredView(THIS^,B_TL_1.IObjectIdentifier);
	3:
		fcXMLStructuredView(THIS^,C_BV_1.IObjectIdentifier);
		fcXMLAddStructuredViewToDevice(THIS^);
	0: 
		usiCreateCase := 1;
ELSE
	usiCreateCase := 0;
END_CASE
END_METHOD

METHOD metCREATE_KBOB_2021_V2 : BOOL;
VAR_INPUT
END_VAR
VAR
	oStatus		:	WagoSysErrorBase.FbResult;
	usiErrors	:	USINT;
END_VAR
(* Resett *)
usiErrors := 0;	

(* Create Objeccts *)
CASE usiCreateCase OF
	1:	
		usiErrors := usiErrors + TO_USINT(NOT metCreate_A_BI_1());
	2:
		usiErrors := usiErrors + TO_USINT(NOT metCreate_B_TL_1());
	3:	
		usiErrors := usiErrors + TO_USINT(NOT metCreate_C_BV_1());
	0: 
		usiCreateCase := 1;
ELSE
	usiCreateCase := 0;
END_CASE;

(* STRUCT VIEW *)
metCREATE_STRUCTVIEW_KBOB_2021_V2();

(* OK = 0*)
metCREATE_KBOB_2021_V2 := NOT TO_BOOL(usiErrors);
END_METHOD

(*FB_Exit muss explizit implementiert werden. Wenn es eine Implementierung gibt, dann wird 
die Methode aufgerufen, bevor die Steuerung den Code der Funktionsbaustein-Instanz entfernt
(impliziter Aufruf. Der Rückgabewert wird nicht ausgewertet.*)
METHOD FB_Exit : BOOL
VAR_INPUT
	(* TRUE: Die Exit-Methode wird aufgerufen, um die Instanz zu verlassen, die hinterher kopiert wird Online-Change).  *)
	bInCopyCode	: BOOL;
END_VAR
(* A_BO_1*)
IF A_BI_1.xIsCreated THEN
	A_BI_1.Delete();	
END_IF;
(* B_TL_1 *)
IF B_TL_1.xIsCreated THEN
	B_TL_1.Delete();
END_IF;
(* C_BV_1 *)
IF C_BV_1.xIsCreated THEN
	C_BV_1.Delete();
END_IF;
END_METHOD

METHOD metCYCLIC_DESCRIPTION_FIX
VAR_INPUT
END_VAR
(* A_BI_1 *)
IF A_BI_1.xIsCreated THEN
	IF A_BI_1.sDescription <> A_BI_1._sDescription THEN
		A_BI_1.sDescription := A_BI_1._sDescription;
	END_IF;
END_IF;

(* B_TL_1 *)
IF B_TL_1.xIsCreated THEN
	IF B_TL_1.sDescription <> B_TL_1._sDescription THEN
		B_TL_1.sDescription := B_TL_1._sDescription;
	END_IF;
END_IF;

(* C_BV_1 *)
IF C_BV_1.xIsCreated THEN
	IF C_BV_1.sDescription <> C_BV_1._sDescription THEN
		C_BV_1.sDescription := C_BV_1._sDescription;
	END_IF;
END_IF;
END_METHOD

METHOD metCYCLIC_KBOB_2017_V1
VAR_INPUT
END_VAR
(* A_BI_1 *)
IF A_BI_1.xIN <> xValue THEN
	A_BI_1.xIN := xValue;				
END_IF;	
(* C_BV_1 *)
IF C_BV_1.xPresentValue <> xError THEN
	C_BV_1.xPresentValue := xError;				
END_IF;
END_METHOD

METHOD metCYCLIC_KBOB_2021_V2
VAR_INPUT
END_VAR
(* A_BI_1 *)
IF A_BI_1.xIN <> xValue THEN
	A_BI_1.xIN := xValue;				
END_IF;	
(* C_BV_1 *)
IF C_BV_1.xPresentValue <> xError THEN
	C_BV_1.xPresentValue := xError;				
END_IF;
END_METHOD

END_FUNCTION_BLOCK

// 30 Program Organization Units/FBs/OBJ_IDENTIFER_BASE/FB_OBJ_ID_BASE
FUNCTION_BLOCK ABSTRACT FB_OBJ_ID_BASE IMPLEMENTS ITF_OBJ_ID_BASE
VAR_INPUT
	ITF_BMK_IN	:	CtaAppBmk.ITF_BMK;
END_VAR
VAR_OUTPUT
END_VAR
VAR
	(*ObjectId*)
	dwOBJ_ID_BASE	:	DWORD;	// 1..4194302
	(* Status *)
	usiCreateCase	:	USINT	:= 1;
	usiErrors		:	USINT;
	xCreatet		:	BOOL;
	xAllowCreate	:	BOOL;
	xAllowDelete	:	BOOL;
	xErrorCreate	:	BOOL;
	xRetry			:	BOOL;
	xRetryed		:	BOOL;
	xDelete			:	BOOL;	
	ITF_NEXT_OBJ	:	ITF_OBJ_ID_BASE;
END_VAR

(* Creat BacNet Objects on Valid ID *)
IF xAllowCreate AND_THEN GVL_BACNET.fbBacNetParameter.proInitDone AND GVL_BACNET.fbBacNetParameter.proCreate AND NOT xCreatet AND NOT xRetryed AND OBJ_ID_BASE <> 0 THEN
	(* Create *)
	xCreatet := metCREATE();
	(* Inkrement usiCreateCase *)
	usiCreateCase := usiCreateCase + 1;
	(* Retry if failed *)
	IF NOT xCreatet AND xErrorCreate THEN
		IF xRetry THEN
			xRetryed := TRUE;
			metDELETE();
		ELSE
			xRetry := TRUE;
		END_IF;
	END_IF;
	xDelete := FALSE;
ELSE
	usiErrors	:= 0;
END_IF;
(* Delete BacNet *)
IF (GVL_BACNET.fbBacNetParameter.proDelete) AND (xCreatet OR xDelete) THEN
	xAllowCreate := FALSE;
	xDelete 	:= metDELETE();
	xCreatet 	:= FALSE;
	(* Reset retry *)
	xRetry 			:= FALSE;
	xRetryed 		:= FALSE;
	xAllowCreate 	:= FALSE;
	xAllowDelete	:= FALSE;
ELSE
	xDelete := FALSE;
END_IF;

PROPERTY OBJ_ID_BASE : DWORD
GET
(* Check if Object ID is 0 *)
IF dwOBJ_ID_BASE = 0 THEN
	IF __QUERYINTERFACE(ITF_BMK_IN,ITF_BMK_IN) THEN
		(* Check if BMK is avaiable *)
		IF NOT ITF_BMK_IN.proNoBmkInList THEN
			(* Calculate Object ID with BMK *)	
			dwOBJ_ID_BASE := fcBmkToAdr(ITF_BMK_IN);
		END_IF;
	END_IF;
ELSE
	(* Take the current Object ID *)
	OBJ_ID_BASE := dwOBJ_ID_BASE;
END_IF;
END_GET
END_PROPERTY

PROPERTY OBJ_NAME_BASE : STRING
GET
OBJ_NAME_BASE := '';
IF __QUERYINTERFACE(ITF_BMK_IN,ITF_BMK_IN) THEN
	(* Check if BMK is avaiable *)
	IF NOT ITF_BMK_IN.proNoBmkInList THEN
		(* Take AKS or BMK as Object Name*)
		IF GVL_BACNET.fbBacNetParameter.proUseAKS THEN
			(* AKS *)
			OBJ_NAME_BASE := ITF_BMK_IN.proGetAKS;
		ELSE
			(* BMK *)
			OBJ_NAME_BASE := ITF_BMK_IN.proGetBMK;
		END_IF;
	END_IF;
END_IF;
END_GET
END_PROPERTY

PROPERTY OBJ_NAME_DESCRIPTION : STRING
GET
OBJ_NAME_DESCRIPTION := '';
IF __QUERYINTERFACE(ITF_BMK_IN,ITF_BMK_IN) THEN
	(* Check if BMK is avaiable *)
	IF NOT ITF_BMK_IN.proNoBmkInList THEN
		(* Get Vendor Name *)
		OBJ_NAME_DESCRIPTION := ITF_BMK_IN.proGetVendorDesignation;
		(* Check if not empty *)
		IF OBJ_NAME_DESCRIPTION <> '' THEN
			(* Add space if no space at the end *)
			IF OBJ_NAME_DESCRIPTION[Standard.LEN(OBJ_NAME_DESCRIPTION)-1] <> TO_BYTE(' ') THEN
				(* Add Space *)
				OBJ_NAME_DESCRIPTION := Standard.CONCAT(OBJ_NAME_DESCRIPTION,' ');
			END_IF;
		END_IF;
	END_IF;
END_IF;
END_GET
END_PROPERTY

METHOD ABSTRACT metCREATE : BOOL;
VAR_INPUT
END_VAR
VAR
END_VAR
END_METHOD

METHOD ABSTRACT metDELETE : BOOL
VAR_INPUT
END_VAR
END_METHOD

//FB_Exit muss explizit implementiert werden. Wenn es eine Implementierung gibt, dann wird 
//die Methode aufgerufen, bevor die Steuerung den Code der Funktionsbaustein-Instanz entfernt
//(impliziter Aufruf. Der Rückgabewert wird nicht ausgewertet.
METHOD FB_Exit: BOOL
VAR_INPUT    
bInCopyCode: BOOL;  // TRUE: Die Exit-Methode wird aufgerufen, um die Instanz zu verlassen, die hinterher kopiert wird Online-Change).  
END_VAR
metDELETE();
END_METHOD

//FB_Init ist immer implizit verfügbar und wird primär für die Initialisierung verwendet.
//Der Rückgabewert wird nicht ausgewertet. Für gezielte Einflussnahme können Sie
//die Methoden explizit deklarieren und darin mit dem Standard-Initialisierungscode 
//zusätzlichen Code bereitstellen. Sie können den Rückgabewert auswerten.
METHOD FB_Init: BOOL
VAR_INPUT    
	bInitRetains: BOOL; // TRUE: Die Retain-Variablen werden initialisiert (Reset warm / Reset kalt)    
	bInCopyCode: BOOL;  // TRUE: Die Instanz wird danach in den Kopiercode kopiert (Online-Change)
END_VAR
VAR
	
END_VAR
GVL_BACNET.fbBacNetParameter.metAddObj(THIS^);
END_METHOD

PROPERTY proINextObj : ITF_OBJ_ID_BASE
SET
ITF_NEXT_OBJ := proINextObj;
END_SET
GET
proINextObj := ITF_NEXT_OBJ;
END_GET
END_PROPERTY

PROPERTY proIsCreatet : BOOL
GET
proIsCreatet := xCreatet OR xRetryed;
END_GET
END_PROPERTY

PROPERTY proAllowCreate : BOOL
SET
xAllowCreate := proAllowCreate;
END_SET
END_PROPERTY

PROPERTY proAllowDelete : BOOL
SET
xAllowDelete := proAllowDelete;
END_SET
END_PROPERTY

END_FUNCTION_BLOCK

// 21 Interface/OBJ_IDENTIFER_BASE/ITF_OBJ_ID_BASE
INTERFACE ITF_OBJ_ID_BASE EXTENDS __SYSTEM.IQueryInterface

//FB_Exit muss explizit implementiert werden. Wenn es eine Implementierung gibt, dann wird 
//die Methode aufgerufen, bevor die Steuerung den Code der Funktionsbaustein-Instanz entfernt
//(impliziter Aufruf. Der Rückgabewert wird nicht ausgewertet.
METHOD FB_Exit: BOOL
VAR_INPUT    
bInCopyCode: BOOL;  // TRUE: Die Exit-Methode wird aufgerufen, um die Instanz zu verlassen, die hinterher kopiert wird Online-Change).  
END_VAR

(* Implement *)
//metDELETE();
END_METHOD

METHOD metCREATE : BOOL;
VAR_INPUT
END_VAR
END_METHOD

PROPERTY OBJ_ID_BASE : DWORD
GET
END_GET
END_PROPERTY

PROPERTY OBJ_NAME_BASE : STRING
GET
END_GET
END_PROPERTY

PROPERTY OBJ_NAME_DESCRIPTION : STRING
GET
END_GET
END_PROPERTY

METHOD metDELETE : BOOL
VAR_INPUT
END_VAR
END_METHOD

PROPERTY proINextObj : ITF_OBJ_ID_BASE
SET
END_SET
GET
END_GET
END_PROPERTY

PROPERTY proAllowCreate : BOOL
SET
END_SET
END_PROPERTY

PROPERTY proIsCreatet : BOOL
GET
END_GET
END_PROPERTY

PROPERTY proAllowDelete : BOOL
SET
END_SET
END_PROPERTY

END_INTERFACE

// 30 Program Organization Units/FCs/BmkToAdr/fcBmkToAdr
FUNCTION fcBmkToAdr : DWORD
VAR_INPUT
	ITF_BMK	:	CtaAppBmk.ITF_BMK;
END_VAR
VAR
	stBMK	:	STRING(7);
	iLen	:	INT;
	wFu		:	WORD;
	wBl		:	WORD;
	wDe		:	WORD;
END_VAR

(* Not Valid *)
fcBmkToAdr := 0;
IF __QUERYINTERFACE(ITF_BMK,ITF_BMK) THEN
	IF ITF_BMK.proGetObjectId <> '' THEN
		stBMK := ITF_BMK.proGetBMK;
		(* Check if Valid BMK min 5 Charakters *)
		IF Standard.LEN(stBMK) >= 5 AND Standard.LEN(stBMK) <= 7 THEN
			iLen := TO_INT(Standard.LEN(stBMK));	
			wFu := TO_WORD(Standard.LEFT(stBMK,TO_INT(-4 + iLen)));
			wBl := TO_WORD(Standard.MID(stBMK,2,(-2 + iLen)));
			wDe := TO_WORD(Standard.RIGHT(stBMK,1));
			(* Check if first Charakters are >= 1 & <= 999*)
			IF wFu >= 1 AND wFu <= 999 THEN
				IF wBl >= 1 AND wBl <= 99 THEN
					IF wDe >= 1 AND wDe <= 2 THEN
						(* Adr 100000 - 297802*)
						fcBmkToAdr := 100000 + ((wFu-1)*198) + ((wBl-1)*2) + ((wDe)*1);
					END_IF;
				END_IF;
			END_IF;
		END_IF;
	END_IF;
END_IF

END_FUNCTION

// 30 Program Organization Units/FCs/XMLFcs/XML BacNet Override/DELETENODE/fcXMLDeleteOverrideNode
FUNCTION fcXMLDeleteOverrideNode : BOOL
VAR_INPUT
	stBacNetIdWithType					:	STRING[8];
END_VAR
VAR
	stBacNetStructView					:	STRING[8];
	stParentPath						:	STRING[80];
	stXmlPath							:	STRING[80];
END_VAR

// xml path
stXmlPath := '/home/user/bacnet/config/override.xml';
// Create BacNet Object 
stParentPath := '';
stParentPath := '//*/objLst';
IF fcXMLDeleteNode(stParentPath,'obj','id',stBacNetIdWithType,'','',stXmlPath) THEN	
	fcXMLDeleteOverrideNode := TRUE;
	GVL_BACNET.fbBacNetParameter.proRebootRequired := TRUE;
END_IF;

END_FUNCTION

// 30 Program Organization Units/FCs/XMLFcs/XMLBase/fcXMLDeleteNode
FUNCTION fcXMLDeleteNode : BOOL
VAR_INPUT
	stParentPath			:	STRING(100);	// Start with '//*/
	stNodeName				:	STRING(100);
	stAttribute1			:	STRING(100);
	stAttribute1Value		:	STRING(150);
	stAttribute2			:	STRING(100);
	stAttribute2Value		:	STRING(150);
	stXmlFilePathName		:	STRING(255);
END_VAR
VAR
	stCommand			:	STRING(1000);
	stTemp				:	STRING(255);
	stResult			:	STRING(255);
	RTS_IEC_RESULT		:	SysTypes.RTS_IEC_RESULT;
END_VAR

IF fcXMLCheckNode(stParentPath,stNodeName,stAttribute1,stAttribute1Value,stAttribute2,stAttribute2Value,stXmlFilePathName) THEN
	stCommand := 	'';
	stTemp	  := 	'';
	stTemp	  :=	'xmlstarlet ed -L -d "';
	StrConcatA(ADR(stTemp),ADR(stCommand),TO_INT(SIZEOF(stCommand)));
	stTemp	  := 	'';
	stTemp	  :=	stParentPath;
	StrConcatA(ADR(stTemp),ADR(stCommand),TO_INT(SIZEOF(stCommand)));
	stTemp	  := 	'';
	stTemp	  :=	'/';
	StrConcatA(ADR(stTemp),ADR(stCommand),TO_INT(SIZEOF(stCommand)));
	stTemp	  := 	'';
	stTemp	  :=	stNodeName;
	StrConcatA(ADR(stTemp),ADR(stCommand),TO_INT(SIZEOF(stCommand)));
	stTemp	  := 	'';
	stTemp	  :=	SEL(stAttribute1 <> '',' ','[@');
	StrConcatA(ADR(stTemp),ADR(stCommand),TO_INT(SIZEOF(stCommand)));
	stTemp	  := 	'';
	stTemp	  :=	stAttribute1;
	StrConcatA(ADR(stTemp),ADR(stCommand),TO_INT(SIZEOF(stCommand)));
	stTemp	  := 	'';
	stTemp	  :=	SEL(stAttribute1 <> '',' ','=$'');
	StrConcatA(ADR(stTemp),ADR(stCommand),TO_INT(SIZEOF(stCommand)));
	stTemp	  := 	'';
	stTemp	  :=	SEL(stAttribute1 <> '','',stAttribute1Value);
	StrConcatA(ADR(stTemp),ADR(stCommand),TO_INT(SIZEOF(stCommand)));
	stTemp	  := 	'';
	stTemp	  :=	SEL(stAttribute1 <> '','',SEL(stAttribute2 <> '','$']','$' and @'));
	StrConcatA(ADR(stTemp),ADR(stCommand),TO_INT(SIZEOF(stCommand)));
	stTemp	  := 	'';
	stTemp	  :=	stAttribute2;
	StrConcatA(ADR(stTemp),ADR(stCommand),TO_INT(SIZEOF(stCommand)));
	stTemp	  := 	'';
	stTemp	  :=	SEL(stAttribute2 <> '',' ','=$'');
	StrConcatA(ADR(stTemp),ADR(stCommand),TO_INT(SIZEOF(stCommand)));
	stTemp	  := 	'';
	stTemp	  :=	SEL(stAttribute2 <> '','',stAttribute2Value);
	StrConcatA(ADR(stTemp),ADR(stCommand),TO_INT(SIZEOF(stCommand)));
	stTemp	  := 	'';
	stTemp	  :=	SEL(stAttribute2 <> '','','$']');
	StrConcatA(ADR(stTemp),ADR(stCommand),TO_INT(SIZEOF(stCommand)));
	stTemp	  := 	'';
	stTemp	  :=	'" ';
	StrConcatA(ADR(stTemp),ADR(stCommand),TO_INT(SIZEOF(stCommand)));
	stTemp	  := 	'';
	stTemp	  :=	stXmlFilePathName;
	StrConcatA(ADR(stTemp),ADR(stCommand),TO_INT(SIZEOF(stCommand)));

	SysProcess_Implementation.SysProcessExecuteCommand(stCommand,ADR(RTS_IEC_RESULT));
	fcXMLDeleteNode := TRUE;
END_IF;

END_FUNCTION

// 30 Program Organization Units/FCs/BacNetId/fcBacNetIdToIdWitType
FUNCTION fcBacNetIdToIdWitType : STRING(8)
VAR_INPUT
	diObjId		:	DINT;
	enObjType	:	WagoTypesBACnet.eBACnetObjectType;
END_VAR
VAR
	dwID		:	DWORD;
END_VAR

dwID := TO_DWORD(diObjId);
dwID.22 := enObjType.0;
dwID.23 := enObjType.1;
dwID.24 := enObjType.2;
dwID.25 := enObjType.3;
dwID.26 := enObjType.4;
dwID.27 := enObjType.5;
dwID.28 := enObjType.6;
dwID.29 := enObjType.7;
dwID.30 := enObjType.8;
dwID.31 := enObjType.9;

fcBacNetIdToIdWitType := fcDWordToHexString(dwID);

END_FUNCTION

// 30 Program Organization Units/FCs/BacNetId/fcDWordToHexString
FUNCTION fcDWordToHexString : STRING[8]
VAR_INPUT
	dwId			:	DWORD;
END_VAR
VAR
	udiData		    :   UDINT;
	udiDiv8         :   UDINT;
	udiDiv7         :   UDINT;
	udiDiv6         :   UDINT;
	udiDiv5         :   UDINT;
    udiDiv4         :   UDINT;
    udiDiv3         :   UDINT;
    udiDiv2         :   UDINT;
    udiDiv1         :   UDINT;
	usiPos8         :   USINT;
	usiPos7         :   USINT;
	usiPos6         :   USINT;
	usiPos5         :   USINT;
    usiPos4         :   USINT;                // 0-F
    usiPos3         :   USINT;                // 0-F
    usiPos2         :   USINT;                // 0-F
    usiPos1         :   USINT;                // 0-F    
    ayOfStr         :   ARRAY[0..15] OF STRING[1] := ['0','1','2','3','4','5','6','7','8','9','A','B','C','D','E','F'];
END_VAR

udiData := DWORD_TO_UDINT(dwId);
IF udiData > 0 THEN
    usiPos8 :=              TO_USINT(                                           (udiData MOD (16)));
    udiDiv8 :=                                  			    (udiData -(udiData MOD (16)))/(16);
    usiPos7 :=              TO_USINT(                                       	(udiDiv8 MOD (16)));
    udiDiv7 :=                                       		  (udiDiv8 - (udiDiv8  MOD (16)))/(16);
    usiPos6 :=              TO_USINT(                                        	(udiDiv7 MOD (16)));
    udiDiv6 :=                     						      (udiDiv7 - (udiDiv7  MOD (16)))/(16);        
    usiPos5 :=              TO_USINT(                                           (udiDiv6 MOD (16)));
    udiDiv5 :=                     						      (udiDiv6 - (udiDiv6  MOD (16)))/(16); 
    usiPos4 :=              TO_USINT(                                           (udiDiv5 MOD (16)));
    udiDiv4 :=                                  			  (udiDiv5 - (udiDiv5  MOD (16)))/(16); 
    usiPos3 :=              TO_USINT(                                       	(udiDiv4 MOD (16)));
    udiDiv3 :=                                       		  (udiDiv4 - (udiDiv4  MOD (16)))/(16);
    usiPos2 :=              TO_USINT(                                        	(udiDiv3 MOD (16)));
    udiDiv2 :=                     						      (udiDiv3 - (udiDiv3  MOD (16)))/(16);        
    usiPos1 :=              TO_USINT(                                           (udiDiv2 MOD (16)));

fcDWordToHexString	 := CONCAT(ayOfStr[usiPos1],
                        CONCAT(ayOfStr[usiPos2],
                        CONCAT(ayOfStr[usiPos3],
                        CONCAT(ayOfStr[usiPos4],
                        CONCAT(ayOfStr[usiPos5],
                        CONCAT(ayOfStr[usiPos6],
						CONCAT(ayOfStr[usiPos7],
                               ayOfStr[usiPos8]


)))))));

ELSE
    fcDWordToHexString := '00000000';
END_IF;

END_FUNCTION

// 30 Program Organization Units/FCs/XMLFcs/XML BacNet Override/STRUCTUREDVIEW/fcXMLDeleteStructuredViewFromDevice
FUNCTION fcXMLDeleteStructuredViewFromDevice : BOOL
VAR_INPUT
	stBacNetIdWithType					:	STRING[8];
END_VAR
VAR
	stBacNetDeviceId					:	STRING[8];
	stParentPath						:	STRING[80];
	stXmlPath							:	STRING[80];
END_VAR

// xml path
stXmlPath := '/home/user/bacnet/config/override.xml';
stBacNetDeviceId 	:= GVL_BACNET.stBacNetDeviceId;
// Create BacNet Object 
stParentPath := '';
stParentPath := CONCAT(CONCAT(CONCAT(CONCAT('//*/objLst/obj[@id=$'',stBacNetDeviceId),'$']/p[@id=$''),TO_STRING(TO_INT(WagoTypesBACnet.eBACnetPropertyIdentifier.PROP_STRUCTURED_OBJECT_LIST))),'$']');	
IF fcXMLDeleteNode(stParentPath,'n','t','192','v',stBacNetIdWithType,stXmlPath) THEN	
	fcXMLDeleteStructuredViewFromDevice := TRUE;
END_IF;

END_FUNCTION

// 30 Program Organization Units/FCs/UTF8Fcs/fcUtfToAscii
FUNCTION fcUtfToAscii : STRING(255)
VAR_INPUT
	stIn	:	STRING(255);
END_VAR
VAR
	iSafety	:	INT;
	iPos	:	INT;
	iLen	:	INT;
END_VAR

IF GVL_BACNET.fbBacNetParameter.fbxAnsiCodiert.proValue THEN
	(* Ä *)
	IF Standard.LEN('Ä') <> 1 THEN	// Check if UTF 8 = 2 Byte or ASCII = 1 Byte
		iSafety := 0;
		WHILE Standard.FIND(stIn,'Ä') <> 0 AND iSafety < 255 DO	
			iPos 		:= Standard.FIND(stIn,'Ä')-1;
			stIn 		:= Standard.DELETE(stIn,Standard.LEN('Ä')-1,Standard.FIND(stIn,'Ä'));
			stIn[iPos]	:= 196;	// ANSI Ä
			iSafety := iSafety + 1;
		END_WHILE;
	END_IF;
	IF Standard.LEN('ä') <> 1 THEN 	// Check if UTF 8 = 2 Byte or ASCII = 1 Byte
		iSafety := 0;
		WHILE Standard.FIND(stIn,'ä') <> 0 AND iSafety < 255 DO	
			iPos 		:= Standard.FIND(stIn,'ä')-1;
			stIn 		:= Standard.DELETE(stIn,Standard.LEN('ä')-1,Standard.FIND(stIn,'ä'));
			stIn[iPos]	:= 228;	// ANSI ä
			iSafety := iSafety + 1;
		END_WHILE;
	END_IF;
	(* Ö *)
	IF Standard.LEN('Ö') <> 1 THEN	// Check if UTF 8 = 2 Byte or ASCII = 1 Byte
		iSafety := 0;
		WHILE Standard.FIND(stIn,'Ö') <> 0 AND iSafety < 255 DO	
			iPos 		:= Standard.FIND(stIn,'Ö')-1;
			stIn 		:= Standard.DELETE(stIn,Standard.LEN('Ö')-1,Standard.FIND(stIn,'Ö'));
			stIn[iPos]	:= 214;	// ANSI Ö
			iSafety := iSafety + 1;
		END_WHILE;
	END_IF;
	IF Standard.LEN('ö') <> 1 THEN	// Check if UTF 8 = 2 Byte or ASCII = 1 Byte
		iSafety := 0;
		WHILE Standard.FIND(stIn,'ö') <> 0 AND iSafety < 255 DO	
			iPos 		:= Standard.FIND(stIn,'ö')-1;
			stIn 		:= Standard.DELETE(stIn,Standard.LEN('ö')-1,Standard.FIND(stIn,'ö'));
			stIn[iPos]	:= 246;	// ANSI ö
			iSafety := iSafety + 1;
		END_WHILE;
	END_IF;
	(* Ü *)
	IF Standard.LEN('Ü') <> 1 THEN	// Check if UTF 8 = 2 Byte or ASCII = 1 Byte
		iSafety := 0;
		WHILE Standard.FIND(stIn,'Ü') <> 0 AND iSafety < 255 DO	
			iPos 		:= Standard.FIND(stIn,'Ü')-1;
			stIn 		:= Standard.DELETE(stIn,Standard.LEN('Ü')-1,Standard.FIND(stIn,'Ü'));
			stIn[iPos]	:= 220;	// ANSI Ü
			iSafety := iSafety + 1;
		END_WHILE;
	END_IF;
	IF Standard.LEN('ü') <> 1 THEN	// Check if UTF 8 = 2 Byte or ASCII = 1 Byte
		iSafety := 0;
		WHILE Standard.FIND(stIn,'ü') <> 0 AND iSafety < 255 DO	
			iPos 		:= Standard.FIND(stIn,'ü')-1;
			stIn 		:= Standard.DELETE(stIn,Standard.LEN('ü')-1,Standard.FIND(stIn,'ü'));
			stIn[iPos]	:= 252;	// ANSI ü
			iSafety := iSafety + 1;
		END_WHILE;
	END_IF;
END_IF;
fcUtfToAscii := stIn;

END_FUNCTION

// 30 Program Organization Units/FCs/BacNetText/fcGetBcText
FUNCTION fcGetBcText : STRING
VAR_INPUT
	stTextListName			:	STRING;
	stTextListAdr			:	STRING;
END_VAR
VAR
END_VAR

fcGetBcText := CmpDynamicText.DynamicTextGetDefaultText(ADR(stTextListName),ADR(stTextListAdr))^;

END_FUNCTION

// 30 Program Organization Units/FCs/XMLFcs/XML BacNet Override/TRENDLOG/fcXMLTrendLogOverride
FUNCTION fcXMLTrendLogOverride : BOOL
VAR_INPUT
	I_BACnetTrendLog_large 				:	WagoTypesBacnet.I_BACnetTrendLog_large;
	I_BACnetTrendLogObjectRef			:	WagoTypesBACnet.I_BACnetObjectIdentifier;
	enTrendLogObjRefPropId				:	WagoTypesBACnet.eBACnetPropertyIdentifier;	
END_VAR
VAR
	stBacNetTrendLogObjId				:	STRING[8];
	stBacNetTrendLogObjRefId			:	STRING[8];	
	stParentPath						:	STRING[80];
	stXmlPath							:	STRING[80];
END_VAR

IF __QUERYINTERFACE(I_BACnetTrendLogObjectRef,I_BACnetTrendLogObjectRef) AND __QUERYINTERFACE(I_BACnetTrendLog_large,I_BACnetTrendLog_large) THEN
	// Get Information
	stBacNetTrendLogObjId 		:= fcBacNetIdToIdWitType(I_BACnetTrendLog_large.IObjectIdentifier.diInstance,I_BACnetTrendLog_large.IObjectIdentifier.eObjectType);
	stBacNetTrendLogObjRefId 	:= fcBacNetIdToIdWitType(I_BACnetTrendLogObjectRef.diInstance,I_BACnetTrendLogObjectRef.eObjectType);
	// xml path
	stXmlPath := '/home/user/bacnet/config/override.xml';
	// Create BacNet Object 
	stParentPath := '';
	stParentPath := '//*/objLst';
	IF fcXMLAddNode(stParentPath,'obj','id',stBacNetTrendLogObjId,'','',stXmlPath,FALSE) THEN	
		fcXMLTrendLogOverride := TRUE;
	END_IF;
	// Create PROP_OBJECT_NAME
	stParentPath := '';
	stParentPath := CONCAT('//*/objLst/obj[@id=$'',CONCAT(stBacNetTrendLogObjId,'$']'));	
	IF fcXMLAddNode(stParentPath,'p','id',TO_STRING(TO_INT(WagoTypesBACnet.eBACnetPropertyIdentifier.PROP_OBJECT_NAME)),'','',stXmlPath,FALSE) THEN	
		fcXMLTrendLogOverride := TRUE;
	END_IF;
		// Create Node PROP_OBJECT_NAME
		stParentPath := '';
		stParentPath := CONCAT(CONCAT(CONCAT(CONCAT('//*/objLst/obj[@id=$'',stBacNetTrendLogObjId),'$']/p[@id=$''),TO_STRING(TO_INT(WagoTypesBACnet.eBACnetPropertyIdentifier.PROP_OBJECT_NAME))),'$']');	
		IF fcXMLAddNode(stParentPath,'n','t','112','v',I_BACnetTrendLog_large.sObjectName,stXmlPath,FALSE) THEN	
			fcXMLTrendLogOverride := TRUE;
		END_IF;
	// Create PROP_OBJECT_IDENTIFIER
	stParentPath := '';
	stParentPath := CONCAT('//*/objLst/obj[@id=$'',CONCAT(stBacNetTrendLogObjId,'$']'));	
	IF fcXMLAddNode(stParentPath,'p','id',TO_STRING(TO_INT(WagoTypesBACnet.eBACnetPropertyIdentifier.PROP_OBJECT_IDENTIFIER)),'','',stXmlPath,FALSE) THEN	
		fcXMLTrendLogOverride := TRUE;
	END_IF;
		// Create Node PROP_OBJECT_IDENTIFIER
		stParentPath := '';
		stParentPath := CONCAT(CONCAT(CONCAT(CONCAT('//*/objLst/obj[@id=$'',stBacNetTrendLogObjId),'$']/p[@id=$''),TO_STRING(TO_INT(WagoTypesBACnet.eBACnetPropertyIdentifier.PROP_OBJECT_IDENTIFIER))),'$']');	
		IF fcXMLAddNode(stParentPath,'n','t','192','v',stBacNetTrendLogObjId,stXmlPath,FALSE) THEN	
			fcXMLTrendLogOverride := TRUE;
		END_IF;
	// Create PROP_RELIABILITY_EVALUATION_INHIBIT
	stParentPath := '';
	stParentPath := CONCAT('//*/objLst/obj[@id=$'',CONCAT(stBacNetTrendLogObjId,'$']'));	
	IF fcXMLAddNode(stParentPath,'p','id',TO_STRING(TO_INT(WagoTypesBACnet.eBACnetPropertyIdentifier.PROP_RELIABILITY_EVALUATION_INHIBIT)),'s','1',stXmlPath,FALSE) THEN	
		fcXMLTrendLogOverride := TRUE;
	END_IF;	
	// Create PROP_EVENT_ALGORITHM_INHIBIT_REF
	stParentPath := '';
	stParentPath := CONCAT('//*/objLst/obj[@id=$'',CONCAT(stBacNetTrendLogObjId,'$']'));	
	IF fcXMLAddNode(stParentPath,'p','id',TO_STRING(TO_INT(WagoTypesBACnet.eBACnetPropertyIdentifier.PROP_EVENT_ALGORITHM_INHIBIT_REF)),'s','1',stXmlPath,FALSE) THEN	
		fcXMLTrendLogOverride := TRUE;
	END_IF;	
	// Create PROP_EVENT_ALGORITHM_INHIBIT
	stParentPath := '';
	stParentPath := CONCAT('//*/objLst/obj[@id=$'',CONCAT(stBacNetTrendLogObjId,'$']'));	
	IF fcXMLAddNode(stParentPath,'p','id',TO_STRING(TO_INT(WagoTypesBACnet.eBACnetPropertyIdentifier.PROP_EVENT_ALGORITHM_INHIBIT)),'s','1',stXmlPath,FALSE) THEN	
		fcXMLTrendLogOverride := TRUE;
	END_IF;	
	// Create PROP_EVENT_DETECTION_ENABLE
	stParentPath := '';
	stParentPath := CONCAT('//*/objLst/obj[@id=$'',CONCAT(stBacNetTrendLogObjId,'$']'));	
	IF fcXMLAddNode(stParentPath,'p','id',TO_STRING(TO_INT(WagoTypesBACnet.eBACnetPropertyIdentifier.PROP_EVENT_DETECTION_ENABLE)),'s','1',stXmlPath,FALSE) THEN	
		fcXMLTrendLogOverride := TRUE;
	END_IF;		
	// Create PROP_EVENT_MESSAGE_TEXTS_CONFIG
	stParentPath := '';
	stParentPath := CONCAT('//*/objLst/obj[@id=$'',CONCAT(stBacNetTrendLogObjId,'$']'));	
	IF fcXMLAddNode(stParentPath,'p','id',TO_STRING(TO_INT(WagoTypesBACnet.eBACnetPropertyIdentifier.PROP_EVENT_MESSAGE_TEXTS_CONFIG)),'s','1',stXmlPath,FALSE) THEN	
		fcXMLTrendLogOverride := TRUE;
	END_IF;		
	// Create PROP_EVENT_MESSAGE_TEXTS
	stParentPath := '';
	stParentPath := CONCAT('//*/objLst/obj[@id=$'',CONCAT(stBacNetTrendLogObjId,'$']'));	
	IF fcXMLAddNode(stParentPath,'p','id',TO_STRING(TO_INT(WagoTypesBACnet.eBACnetPropertyIdentifier.PROP_EVENT_MESSAGE_TEXTS)),'','',stXmlPath,FALSE) THEN	
		fcXMLTrendLogOverride := TRUE;
	END_IF;		
	// Create PROP_TRIGGER
	stParentPath := '';
	stParentPath := CONCAT('//*/objLst/obj[@id=$'',CONCAT(stBacNetTrendLogObjId,'$']'));	
	IF fcXMLAddNode(stParentPath,'p','id',TO_STRING(TO_INT(WagoTypesBACnet.eBACnetPropertyIdentifier.PROP_TRIGGER)),'','',stXmlPath,FALSE) THEN	
		fcXMLTrendLogOverride := TRUE;
	END_IF;			
	// Create PROP_INTERVAL_OFFSET
	stParentPath := '';
	stParentPath := CONCAT('//*/objLst/obj[@id=$'',CONCAT(stBacNetTrendLogObjId,'$']'));	
	IF fcXMLAddNode(stParentPath,'p','id',TO_STRING(TO_INT(WagoTypesBACnet.eBACnetPropertyIdentifier.PROP_INTERVAL_OFFSET)),'s','1',stXmlPath,FALSE) THEN	
		fcXMLTrendLogOverride := TRUE;
	END_IF;	
	// Create PROP_ALIGN_INTERVALS
	stParentPath := '';
	stParentPath := CONCAT('//*/objLst/obj[@id=$'',CONCAT(stBacNetTrendLogObjId,'$']'));	
	IF fcXMLAddNode(stParentPath,'p','id',TO_STRING(TO_INT(WagoTypesBACnet.eBACnetPropertyIdentifier.PROP_ALIGN_INTERVALS)),'s','1',stXmlPath,FALSE) THEN	
		fcXMLTrendLogOverride := TRUE;
	END_IF;	
	// Create PROP_LAST_NOTIFY_RECORD
	stParentPath := '';
	stParentPath := CONCAT('//*/objLst/obj[@id=$'',CONCAT(stBacNetTrendLogObjId,'$']'));	
	IF fcXMLAddNode(stParentPath,'p','id',TO_STRING(TO_INT(WagoTypesBACnet.eBACnetPropertyIdentifier.PROP_LAST_NOTIFY_RECORD)),'s','1',stXmlPath,FALSE) THEN	
		fcXMLTrendLogOverride := TRUE;
	END_IF;	
	// Create PROP_RECORDS_SINCE_NOTIFICATION
	stParentPath := '';
	stParentPath := CONCAT('//*/objLst/obj[@id=$'',CONCAT(stBacNetTrendLogObjId,'$']'));	
	IF fcXMLAddNode(stParentPath,'p','id',TO_STRING(TO_INT(WagoTypesBACnet.eBACnetPropertyIdentifier.PROP_RECORDS_SINCE_NOTIFICATION)),'s','1',stXmlPath,FALSE) THEN	
		fcXMLTrendLogOverride := TRUE;
	END_IF;	
	// Create PROP_NOTIFICATION_THRESHOLD
	stParentPath := '';
	stParentPath := CONCAT('//*/objLst/obj[@id=$'',CONCAT(stBacNetTrendLogObjId,'$']'));	
	IF fcXMLAddNode(stParentPath,'p','id',TO_STRING(TO_INT(WagoTypesBACnet.eBACnetPropertyIdentifier.PROP_NOTIFICATION_THRESHOLD)),'s','1',stXmlPath,FALSE) THEN	
		fcXMLTrendLogOverride := TRUE;
	END_IF;	
	// Create PROP_LOG_INTERVAL
	stParentPath := '';
	stParentPath := CONCAT('//*/objLst/obj[@id=$'',CONCAT(stBacNetTrendLogObjId,'$']'));	
	IF fcXMLAddNode(stParentPath,'p','id',TO_STRING(TO_INT(WagoTypesBACnet.eBACnetPropertyIdentifier.PROP_LOG_INTERVAL)),'s','1',stXmlPath,FALSE) THEN	
		fcXMLTrendLogOverride := TRUE;
	END_IF;	
		// Create Node PROP_LOG_INTERVAL
		stParentPath := '';
		stParentPath := CONCAT(CONCAT(CONCAT(CONCAT('//*/objLst/obj[@id=$'',stBacNetTrendLogObjId),'$']/p[@id=$''),TO_STRING(TO_INT(WagoTypesBACnet.eBACnetPropertyIdentifier.PROP_LOG_INTERVAL))),'$']');
		IF fcXMLAddNode(stParentPath,'n','t','32','v','1000',stXmlPath,FALSE) THEN	
			fcXMLTrendLogOverride := TRUE;
		END_IF;
	// Create PROP_LOGGING_TYPE
	stParentPath := '';
	stParentPath := CONCAT('//*/objLst/obj[@id=$'',CONCAT(stBacNetTrendLogObjId,'$']'));	
	IF fcXMLAddNode(stParentPath,'p','id',TO_STRING(TO_INT(WagoTypesBACnet.eBACnetPropertyIdentifier.PROP_LOGGING_TYPE)),'s','1',stXmlPath,FALSE) THEN	
		fcXMLTrendLogOverride := TRUE;
	END_IF;	
		// Create Node PROP_LOGGING_TYPE
		stParentPath := '';
		stParentPath := CONCAT(CONCAT(CONCAT(CONCAT('//*/objLst/obj[@id=$'',stBacNetTrendLogObjId),'$']/p[@id=$''),TO_STRING(TO_INT(WagoTypesBACnet.eBACnetPropertyIdentifier.PROP_LOGGING_TYPE))),'$']');
		IF fcXMLAddNode(stParentPath,'n','t','144','v',TO_STRING(TO_INT(WagoTypesBACnet.eBACnetLoggingType.LOGGING_TYPE_POLLED)),stXmlPath,FALSE) THEN	
			fcXMLTrendLogOverride := TRUE;
		END_IF;		
	// Create PROP_CLIENT_COV_INCREMENT
	stParentPath := '';
	stParentPath := CONCAT('//*/objLst/obj[@id=$'',CONCAT(stBacNetTrendLogObjId,'$']'));	
	IF fcXMLAddNode(stParentPath,'p','id',TO_STRING(TO_INT(WagoTypesBACnet.eBACnetPropertyIdentifier.PROP_CLIENT_COV_INCREMENT)),'s','1',stXmlPath,FALSE) THEN	
		fcXMLTrendLogOverride := TRUE;
	END_IF;	
		// Create Node 276 PROP_CLIENT_COV_INCREMENT
		stParentPath := '';
		stParentPath := CONCAT(CONCAT(CONCAT(CONCAT('//*/objLst/obj[@id=$'',stBacNetTrendLogObjId),'$']/p[@id=$''),TO_STRING(TO_INT(WagoTypesBACnet.eBACnetPropertyIdentifier.PROP_CLIENT_COV_INCREMENT))),'$']');
		IF fcXMLAddNode(stParentPath,'n','t','276','','',stXmlPath,FALSE) THEN	
			fcXMLTrendLogOverride := TRUE;
		END_IF;		
			// Create Node 64 PROP_CLIENT_COV_INCREMENT
			stParentPath := '';
			stParentPath := CONCAT(CONCAT(CONCAT(CONCAT('//*/objLst/obj[@id=$'',stBacNetTrendLogObjId),'$']/p[@id=$''),TO_STRING(TO_INT(WagoTypesBACnet.eBACnetPropertyIdentifier.PROP_CLIENT_COV_INCREMENT))),'$']/n[@t=$'276$']');
			IF fcXMLAddNode(stParentPath,'n','t','64','v','0.1',stXmlPath,FALSE) THEN	
				fcXMLTrendLogOverride := TRUE;
			END_IF;	
	// Create PROP_LOG_DEVICE_OBJ_PROP
	stParentPath := '';
	stParentPath := CONCAT('//*/objLst/obj[@id=$'',CONCAT(stBacNetTrendLogObjId,'$']'));	
	IF fcXMLAddNode(stParentPath,'p','id',TO_STRING(TO_INT(WagoTypesBACnet.eBACnetPropertyIdentifier.PROP_LOG_DEVICE_OBJ_PROP)),'s','1',stXmlPath,FALSE) THEN	
		fcXMLTrendLogOverride := TRUE;
	END_IF;			
		// Create Node 275 PROP_LOG_DEVICE_OBJ_PROP
		stParentPath := '';
		stParentPath := CONCAT(CONCAT(CONCAT(CONCAT('//*/objLst/obj[@id=$'',stBacNetTrendLogObjId),'$']/p[@id=$''),TO_STRING(TO_INT(WagoTypesBACnet.eBACnetPropertyIdentifier.PROP_LOG_DEVICE_OBJ_PROP))),'$']');
		IF fcXMLAddNode(stParentPath,'n','t','275','','',stXmlPath,FALSE) THEN	
			fcXMLTrendLogOverride := TRUE;
		END_IF;
			// Create Node 192 PROP_LOG_DEVICE_OBJ_PROP
			stParentPath := '';
			stParentPath := CONCAT(CONCAT(CONCAT(CONCAT('//*/objLst/obj[@id=$'',stBacNetTrendLogObjId),'$']/p[@id=$''),TO_STRING(TO_INT(WagoTypesBACnet.eBACnetPropertyIdentifier.PROP_LOG_DEVICE_OBJ_PROP))),'$']/n[@t=$'275$']');	
			IF fcXMLAddNode(stParentPath,'n','t','192','v',stBacNetTrendLogObjRefId,stXmlPath,FALSE) THEN	
				fcXMLTrendLogOverride := TRUE;
			ELSE
				fcXMLUpdateAttribute(stParentPath,'n','t','192','v',stBacNetTrendLogObjRefId,stXmlPath);
			END_IF;
			// Create Node 144 PROP_LOG_DEVICE_OBJ_PROP
			stParentPath := '';
			stParentPath := CONCAT(CONCAT(CONCAT(CONCAT('//*/objLst/obj[@id=$'',stBacNetTrendLogObjId),'$']/p[@id=$''),TO_STRING(TO_INT(WagoTypesBACnet.eBACnetPropertyIdentifier.PROP_LOG_DEVICE_OBJ_PROP))),'$']/n[@t=$'275$']');	
			IF fcXMLAddNode(stParentPath,'n','t','144','v',TO_STRING(TO_INT(enTrendLogObjRefPropId)),stXmlPath,FALSE) THEN	
				fcXMLTrendLogOverride := TRUE;
			END_IF;	
	// Create PROP_EVENT_TIME_STAMPS
	stParentPath := '';
	stParentPath := CONCAT('//*/objLst/obj[@id=$'',CONCAT(stBacNetTrendLogObjId,'$']'));	
	IF fcXMLAddNode(stParentPath,'p','id',TO_STRING(TO_INT(WagoTypesBACnet.eBACnetPropertyIdentifier.PROP_EVENT_TIME_STAMPS)),'','',stXmlPath,FALSE) THEN	
		fcXMLTrendLogOverride := TRUE;
	END_IF;
	// Create PROP_COV_RESUBSCRIBE_INTERVAL
	stParentPath := '';
	stParentPath := CONCAT('//*/objLst/obj[@id=$'',CONCAT(stBacNetTrendLogObjId,'$']'));	
	IF fcXMLAddNode(stParentPath,'p','id',TO_STRING(TO_INT(WagoTypesBACnet.eBACnetPropertyIdentifier.PROP_COV_RESUBSCRIBE_INTERVAL)),'s','1',stXmlPath,FALSE) THEN	
		fcXMLTrendLogOverride := TRUE;
	END_IF;	
	// Create PROP_CLIENT_COV_INCREMENT
	stParentPath := '';
	stParentPath := CONCAT('//*/objLst/obj[@id=$'',CONCAT(stBacNetTrendLogObjId,'$']'));	
	IF fcXMLAddNode(stParentPath,'p','id',TO_STRING(TO_INT(WagoTypesBACnet.eBACnetPropertyIdentifier.PROP_CLIENT_COV_INCREMENT)),'s','1',stXmlPath,FALSE) THEN	
		fcXMLTrendLogOverride := TRUE;
	END_IF;	
	// Create PROP_BUFFER_SIZE
	stParentPath := '';
	stParentPath := CONCAT('//*/objLst/obj[@id=$'',CONCAT(stBacNetTrendLogObjId,'$']'));	
	IF fcXMLAddNode(stParentPath,'p','id',TO_STRING(TO_INT(WagoTypesBACnet.eBACnetPropertyIdentifier.PROP_BUFFER_SIZE)),'s','1',stXmlPath,FALSE) THEN	
		fcXMLTrendLogOverride := TRUE;
	END_IF;		
		// Create Node 32 PROP_BUFFER_SIZE
		stParentPath := '';
		stParentPath := CONCAT(CONCAT(CONCAT(CONCAT('//*/objLst/obj[@id=$'',stBacNetTrendLogObjId),'$']/p[@id=$''),TO_STRING(TO_INT(WagoTypesBACnet.eBACnetPropertyIdentifier.PROP_BUFFER_SIZE))),'$']');
		IF fcXMLAddNode(stParentPath,'n','t','32','v','100',stXmlPath,FALSE) THEN	
			fcXMLTrendLogOverride := TRUE;
		END_IF;	
	// Create PROP_RELIABILITY
	stParentPath := '';
	stParentPath := CONCAT('//*/objLst/obj[@id=$'',CONCAT(stBacNetTrendLogObjId,'$']'));	
	IF fcXMLAddNode(stParentPath,'p','id',TO_STRING(TO_INT(WagoTypesBACnet.eBACnetPropertyIdentifier.PROP_RELIABILITY)),'s','0',stXmlPath,FALSE) THEN	
		fcXMLTrendLogOverride := TRUE;
	END_IF;	
	// Create PROP_NOTIFY_TYPE
	stParentPath := '';
	stParentPath := CONCAT('//*/objLst/obj[@id=$'',CONCAT(stBacNetTrendLogObjId,'$']'));	
	IF fcXMLAddNode(stParentPath,'p','id',TO_STRING(TO_INT(WagoTypesBACnet.eBACnetPropertyIdentifier.PROP_NOTIFY_TYPE)),'s','1',stXmlPath,FALSE) THEN	
		fcXMLTrendLogOverride := TRUE;
	END_IF;	
	// Create PROP_EVENT_ENABLE
	stParentPath := '';
	stParentPath := CONCAT('//*/objLst/obj[@id=$'',CONCAT(stBacNetTrendLogObjId,'$']'));	
	IF fcXMLAddNode(stParentPath,'p','id',TO_STRING(TO_INT(WagoTypesBACnet.eBACnetPropertyIdentifier.PROP_EVENT_ENABLE)),'s','1',stXmlPath,FALSE) THEN	
		fcXMLTrendLogOverride := TRUE;
	END_IF;	
	// Create PROP_DESCRIPTION
	stParentPath := '';
	stParentPath := CONCAT('//*/objLst/obj[@id=$'',CONCAT(stBacNetTrendLogObjId,'$']'));	
	IF fcXMLAddNode(stParentPath,'p','id',TO_STRING(TO_INT(WagoTypesBACnet.eBACnetPropertyIdentifier.PROP_DESCRIPTION)),'s','1',stXmlPath,FALSE) THEN	
		fcXMLTrendLogOverride := TRUE;
	END_IF;	
	// Create PROP_NOTIFICATION_CLASS
	stParentPath := '';
	stParentPath := CONCAT('//*/objLst/obj[@id=$'',CONCAT(stBacNetTrendLogObjId,'$']'));	
	IF fcXMLAddNode(stParentPath,'p','id',TO_STRING(TO_INT(WagoTypesBACnet.eBACnetPropertyIdentifier.PROP_NOTIFICATION_CLASS)),'s','1',stXmlPath,FALSE) THEN	
		fcXMLTrendLogOverride := TRUE;
	END_IF;	
	// Create PROP_ACKED_TRANSITIONS
	stParentPath := '';
	stParentPath := CONCAT('//*/objLst/obj[@id=$'',CONCAT(stBacNetTrendLogObjId,'$']'));	
	IF fcXMLAddNode(stParentPath,'p','id',TO_STRING(TO_INT(WagoTypesBACnet.eBACnetPropertyIdentifier.PROP_ACKED_TRANSITIONS)),'','',stXmlPath,FALSE) THEN	
		fcXMLTrendLogOverride := TRUE;
	END_IF;	
	// Set Reboot Required	
	IF fcXMLTrendLogOverride THEN
		GVL_BACNET.fbBacNetParameter.proRebootRequired := TRUE;
	END_IF;	
END_IF;

END_FUNCTION

// 30 Program Organization Units/FCs/XMLFcs/XMLBase/fcXMLAddNode
FUNCTION fcXMLAddNode : BOOL
VAR_INPUT
	stParentPath			:	STRING(100);	// Start with '//*/
	stNodeName				:	STRING(100);
	stAttribute1			:	STRING(100);
	stAttribute1Value		:	STRING(150);
	stAttribute2			:	STRING(100);
	stAttribute2Value		:	STRING(150);
	stXmlFilePathName		:	STRING(255);
	xIgnoreCheck			:	BOOL;
END_VAR
VAR
	stCommand			:	STRING(1000);
	stTemp				:	STRING(255);
	stResult			:	STRING(255);
	RTS_IEC_RESULT		:	SysTypes.RTS_IEC_RESULT;
END_VAR

fcXMLAddNode := FALSE;
IF NOT fcXMLCheckNode(stParentPath,stNodeName,stAttribute1,stAttribute1Value,stAttribute2,stAttribute2Value,stXmlFilePathName) OR xIgnoreCheck THEN
	// Create Node if not exist
	stCommand := 	'';
	stTemp	  := 	'';
	stTemp	  :=	'xmlstarlet ed -L -s "';
	StrConcatA(ADR(stTemp),ADR(stCommand),TO_INT(SIZEOF(stCommand)));
	stTemp	  := 	'';
	stTemp	  :=	stParentPath;
	StrConcatA(ADR(stTemp),ADR(stCommand),TO_INT(SIZEOF(stCommand)));	
	stTemp	  := 	'';
	stTemp	  :=	'" -t elem -n "';
	StrConcatA(ADR(stTemp),ADR(stCommand),TO_INT(SIZEOF(stCommand)));		
	stTemp	  := 	'';
	stTemp	  :=	stNodeName;
	StrConcatA(ADR(stTemp),ADR(stCommand),TO_INT(SIZEOF(stCommand)));
	stTemp	  := 	'';
	stTemp	  :=	'" -v "" ';
	StrConcatA(ADR(stTemp),ADR(stCommand),TO_INT(SIZEOF(stCommand)));
	stTemp	  := 	'';
	stTemp	  :=	stXmlFilePathName;
	StrConcatA(ADR(stTemp),ADR(stCommand),TO_INT(SIZEOF(stCommand)));
					
	SysProcess_Implementation.SysProcessExecuteCommand2(stCommand,stResult,SIZEOF(stResult),ADR(RTS_IEC_RESULT));
	
	IF stAttribute1 <> '' THEN
		fcXMLAddAttribute(stParentPath,stNodeName,stAttribute1,stAttribute1Value,'','',stXmlFilePathName,xIgnoreCheck);
	END_IF
	IF stAttribute2 <> '' THEN
		fcXMLAddAttribute(stParentPath,stNodeName,stAttribute2,stAttribute2Value,stAttribute1,stAttribute1Value,stXmlFilePathName,xIgnoreCheck);
	END_IF;
	fcXMLAddNode := TRUE;
END_IF;

END_FUNCTION

// 30 Program Organization Units/FCs/XMLFcs/XMLBase/fcXMLUpdateAttribute
FUNCTION fcXMLUpdateAttribute : BOOL
VAR_INPUT
	stParentPath			:	STRING(100);	// Start with '//*/
	stNodeName				:	STRING(100);
	stAttribute1			:	STRING(100);
	stAttribute1Value		:	STRING(150);
	stAttribute2Uppdate		:	STRING(100);
	stAttribute2ValueUpdate	:	STRING(150);
	stXmlFilePathName		:	STRING(255);
END_VAR
VAR
	stCommand			:	STRING(1000);
	stTemp				:	STRING(255);
	RTS_IEC_RESULT		:	SysTypes.RTS_IEC_RESULT;
END_VAR

stCommand := 	'';
stTemp	  := 	'';
stTemp	  :=	'xmlstarlet ed -L --update "';
StrConcatA(ADR(stTemp),ADR(stCommand),TO_INT(SIZEOF(stCommand)));
stTemp	  := 	'';
stTemp	  :=	stParentPath;
StrConcatA(ADR(stTemp),ADR(stCommand),TO_INT(SIZEOF(stCommand)));
stTemp	  := 	'';
stTemp	  :=	'/';
StrConcatA(ADR(stTemp),ADR(stCommand),TO_INT(SIZEOF(stCommand)));
stTemp	  := 	'';
stTemp	  :=	stNodeName;
StrConcatA(ADR(stTemp),ADR(stCommand),TO_INT(SIZEOF(stCommand)));
stTemp	  := 	'';
stTemp	  :=	SEL(stAttribute1 <> '','','[@');
StrConcatA(ADR(stTemp),ADR(stCommand),TO_INT(SIZEOF(stCommand)));
stTemp	  := 	'';
stTemp	  :=	SEL(stAttribute1 <> '','',stAttribute1);
StrConcatA(ADR(stTemp),ADR(stCommand),TO_INT(SIZEOF(stCommand)));
stTemp	  := 	'';
stTemp	  :=	SEL(stAttribute1 <> '','','=$'');
StrConcatA(ADR(stTemp),ADR(stCommand),TO_INT(SIZEOF(stCommand)));
stTemp	  := 	'';
stTemp	  :=	SEL(stAttribute1 <> '','',stAttribute1Value);
StrConcatA(ADR(stTemp),ADR(stCommand),TO_INT(SIZEOF(stCommand)));
stTemp	  := 	'';
stTemp	  :=	SEL(stAttribute1 <> '','','$']');
StrConcatA(ADR(stTemp),ADR(stCommand),TO_INT(SIZEOF(stCommand)));
stTemp	  := 	'';
stTemp	  :=	'/@';
StrConcatA(ADR(stTemp),ADR(stCommand),TO_INT(SIZEOF(stCommand)));
stTemp	  := 	'';
stTemp	  :=	stAttribute2Uppdate;
StrConcatA(ADR(stTemp),ADR(stCommand),TO_INT(SIZEOF(stCommand)));
stTemp	  := 	'';
stTemp	  :=	'" -v "';
StrConcatA(ADR(stTemp),ADR(stCommand),TO_INT(SIZEOF(stCommand)));
stTemp	  := 	'';
stTemp	  :=	stAttribute2ValueUpdate;
StrConcatA(ADR(stTemp),ADR(stCommand),TO_INT(SIZEOF(stCommand)));
stTemp	  := 	'';
stTemp	  :=	'" ';
StrConcatA(ADR(stTemp),ADR(stCommand),TO_INT(SIZEOF(stCommand)));
stTemp	  := 	'';
stTemp	  :=	stXmlFilePathName;
StrConcatA(ADR(stTemp),ADR(stCommand),TO_INT(SIZEOF(stCommand)));

SysProcess_Implementation.SysProcessExecuteCommand(stCommand,ADR(RTS_IEC_RESULT));

END_FUNCTION

// 30 Program Organization Units/FCs/XMLFcs/XML BacNet Override/STRUCTUREDVIEW/fcXMLStructuredView
FUNCTION fcXMLStructuredView : BOOL
VAR_INPUT
	ITF_OBJ_ID_BASE_IN 					:	ITF_OBJ_ID_BASE;
	I_BACnetStructObjectRef				:	WagoTypesBACnet.I_BACnetObjectIdentifier;
END_VAR
VAR
	stBacNetStructView					:	STRING[8];
	stBacNetObjRefId			:	STRING[8];	
	stParentPath						:	STRING[80];
	stXmlPath							:	STRING[80];
END_VAR

IF __QUERYINTERFACE(I_BACnetStructObjectRef,I_BACnetStructObjectRef) AND __QUERYINTERFACE(ITF_OBJ_ID_BASE_IN,ITF_OBJ_ID_BASE_IN) THEN
	// Get Information
	stBacNetStructView	:= fcBacNetIdToIdWitType(TO_DINT(CONCAT(TO_STRING(ITF_OBJ_ID_BASE_IN.OBJ_ID_BASE),'1')),WagoTypesBacNet.eBACnetObjectType.BACnet_structured_view);
	stBacNetObjRefId 	:= fcBacNetIdToIdWitType(I_BACnetStructObjectRef.diInstance,I_BACnetStructObjectRef.eObjectType);
	// xml path
	stXmlPath := '/home/user/bacnet/config/override.xml';
	// Create BacNet Object 
	stParentPath := '';
	stParentPath := '//*/objLst';
	IF fcXMLAddNode(stParentPath,'obj','id',stBacNetStructView,'','',stXmlPath,FALSE) THEN	
		fcXMLStructuredView := TRUE;
	END_IF;
	// Create PROP_SUBORDINATE_LIST
	stParentPath := '';
	stParentPath := CONCAT('//*/objLst/obj[@id=$'',CONCAT(stBacNetStructView,'$']'));	
	IF fcXMLAddNode(stParentPath,'p','id',TO_STRING(TO_INT(WagoTypesBACnet.eBACnetPropertyIdentifier.PROP_SUBORDINATE_LIST)),'s','1',stXmlPath,FALSE) THEN	
		fcXMLStructuredView := TRUE;
	END_IF;
		// Check if Object Reference Node Exist
		stParentPath := '';
		stParentPath := CONCAT(CONCAT(CONCAT(CONCAT('//*/objLst/obj[@id=$'',stBacNetStructView),'$']/p[@id=$''),TO_STRING(TO_INT(WagoTypesBACnet.eBACnetPropertyIdentifier.PROP_SUBORDINATE_LIST))),'$']/n[@t=$'288$']');			
		IF NOT fcXMLCheckNode(stParentPath,'n','t','192','v',stBacNetObjRefId,stXmlPath) THEN
			// Create Node 288 PROP_SUBORDINATE_LIST
			stParentPath := '';
			stParentPath := CONCAT(CONCAT(CONCAT(CONCAT('//*/objLst/obj[@id=$'',stBacNetStructView),'$']/p[@id=$''),TO_STRING(TO_INT(WagoTypesBACnet.eBACnetPropertyIdentifier.PROP_SUBORDINATE_LIST))),'$']');	
			IF fcXMLAddNode(stParentPath,'n','t','288','','',stXmlPath,TRUE) THEN	
				fcXMLStructuredView := TRUE;
			END_IF;
				// Create Node 192 PROP_SUBORDINATE_LIST
				stParentPath := '';
				stParentPath := CONCAT(CONCAT(CONCAT(CONCAT('//*/objLst/obj[@id=$'',stBacNetStructView),'$']/p[@id=$''),TO_STRING(TO_INT(WagoTypesBACnet.eBACnetPropertyIdentifier.PROP_SUBORDINATE_LIST))),'$']/n[last()]');
				IF fcXMLAddNode(stParentPath,'n','t','192','v',stBacNetObjRefId,stXmlPath,TRUE) THEN	
					fcXMLStructuredView := TRUE;
				END_IF;
		END_IF;
	// Create PROP_OBJECT_NAME
	stParentPath := '';
	stParentPath := CONCAT('//*/objLst/obj[@id=$'',CONCAT(stBacNetStructView,'$']'));	
	IF fcXMLAddNode(stParentPath,'p','id',TO_STRING(TO_INT(WagoTypesBACnet.eBACnetPropertyIdentifier.PROP_OBJECT_NAME)),'','',stXmlPath,FALSE) THEN	
		fcXMLStructuredView := TRUE;
	END_IF;
		// Create Node PROP_OBJECT_NAME
		stParentPath := '';
		stParentPath := CONCAT(CONCAT(CONCAT(CONCAT('//*/objLst/obj[@id=$'',stBacNetStructView),'$']/p[@id=$''),TO_STRING(TO_INT(WagoTypesBACnet.eBACnetPropertyIdentifier.PROP_OBJECT_NAME))),'$']');	
		IF fcXMLAddNode(stParentPath,'n','t','112','v',ITF_OBJ_ID_BASE_IN.OBJ_NAME_BASE,stXmlPath,FALSE) THEN	
			fcXMLStructuredView := TRUE;
		END_IF;
	// Create PROP_OBJECT_IDENTIFIER
	stParentPath := '';
	stParentPath := CONCAT('//*/objLst/obj[@id=$'',CONCAT(stBacNetStructView,'$']'));	
	IF fcXMLAddNode(stParentPath,'p','id',TO_STRING(TO_INT(WagoTypesBACnet.eBACnetPropertyIdentifier.PROP_OBJECT_IDENTIFIER)),'','',stXmlPath,FALSE) THEN	
		fcXMLStructuredView := TRUE;
	END_IF;
		// Create Node PROP_OBJECT_IDENTIFIER
		stParentPath := '';
		stParentPath := CONCAT(CONCAT(CONCAT(CONCAT('//*/objLst/obj[@id=$'',stBacNetStructView),'$']/p[@id=$''),TO_STRING(TO_INT(WagoTypesBACnet.eBACnetPropertyIdentifier.PROP_OBJECT_IDENTIFIER))),'$']');	
		IF fcXMLAddNode(stParentPath,'n','t','192','v',stBacNetStructView,stXmlPath,FALSE) THEN	
			fcXMLStructuredView := TRUE;
		END_IF;		
	// Create PROP_DESCRIPTION
	stParentPath := '';
	stParentPath := CONCAT('//*/objLst/obj[@id=$'',CONCAT(stBacNetStructView,'$']'));	
	IF fcXMLAddNode(stParentPath,'p','id',TO_STRING(TO_INT(WagoTypesBACnet.eBACnetPropertyIdentifier.PROP_DESCRIPTION)),'s','1',stXmlPath,FALSE) THEN	
		fcXMLStructuredView := TRUE;
	END_IF;		
		// Create Node 112 PROP_DESCRIPTION
		stParentPath := '';
		stParentPath := CONCAT(CONCAT(CONCAT(CONCAT('//*/objLst/obj[@id=$'',stBacNetStructView),'$']/p[@id=$''),TO_STRING(TO_INT(WagoTypesBACnet.eBACnetPropertyIdentifier.PROP_DESCRIPTION))),'$']');	
		IF fcXMLAddNode(stParentPath,'n','t','112','v',ITF_OBJ_ID_BASE_IN.OBJ_NAME_DESCRIPTION,stXmlPath,FALSE) THEN	
			fcXMLStructuredView := TRUE;
		END_IF;
	// Create PROP_NODE_SUBTYPE
	stParentPath := '';
	stParentPath := CONCAT('//*/objLst/obj[@id=$'',CONCAT(stBacNetStructView,'$']'));	
	IF fcXMLAddNode(stParentPath,'p','id',TO_STRING(TO_INT(WagoTypesBACnet.eBACnetPropertyIdentifier.PROP_NODE_SUBTYPE)),'s','1',stXmlPath,FALSE) THEN	
		fcXMLStructuredView := TRUE;
	END_IF;	
	// Create PROP_NODE_SUBTYPE
	stParentPath := '';
	stParentPath := CONCAT('//*/objLst/obj[@id=$'',CONCAT(stBacNetStructView,'$']'));	
	IF fcXMLAddNode(stParentPath,'p','id',TO_STRING(TO_INT(WagoTypesBACnet.eBACnetPropertyIdentifier.PROP_NODE_TYPE)),'s','1',stXmlPath,FALSE) THEN	
		fcXMLStructuredView := TRUE;
	END_IF;	
		// Create Node PROP_NODE_SUBTYPE
		stParentPath := '';
		stParentPath := CONCAT(CONCAT(CONCAT(CONCAT('//*/objLst/obj[@id=$'',stBacNetStructView),'$']/p[@id=$''),TO_STRING(TO_INT(WagoTypesBACnet.eBACnetPropertyIdentifier.PROP_NODE_TYPE))),'$']');	
		IF fcXMLAddNode(stParentPath,'n','t','144','v','17',stXmlPath,FALSE) THEN	
			fcXMLStructuredView := TRUE;
		END_IF;	
	// Set Reboot Required	
	IF fcXMLStructuredView THEN
		GVL_BACNET.fbBacNetParameter.proRebootRequired := TRUE;
	END_IF;	
END_IF;

END_FUNCTION

// 30 Program Organization Units/FCs/XMLFcs/XML BacNet Override/STRUCTUREDVIEW/fcXMLAddStructuredViewToDevice
FUNCTION fcXMLAddStructuredViewToDevice : BOOL
VAR_INPUT
	ITF_OBJ_ID_BASE_IN 					:	ITF_OBJ_ID_BASE;
END_VAR
VAR
	stBacNetStructView					:	STRING[8];
	stBacNetDeviceId					:	STRING[8];	
	stParentPath						:	STRING[80];
	stXmlPath							:	STRING[80];
END_VAR

IF __QUERYINTERFACE(ITF_OBJ_ID_BASE_IN,ITF_OBJ_ID_BASE_IN) THEN
	// Get Information
	stBacNetStructView	:= fcBacNetIdToIdWitType(TO_DINT(CONCAT(TO_STRING(ITF_OBJ_ID_BASE_IN.OBJ_ID_BASE),'1')),WagoTypesBacNet.eBACnetObjectType.BACnet_structured_view);
	stBacNetDeviceId 	:= GVL_BACNET.stBacNetDeviceId;
	// xml path
	stXmlPath := '/home/user/bacnet/config/override.xml'; 
	// Create BacNet Device Object 
	stParentPath := '';
	stParentPath := '//*/objLst';
	fcXMLAddNode(stParentPath,'obj','id',stBacNetDeviceId,'','',stXmlPath,FALSE);	
	// Create PROP_STRUCTURED_OBJECT_LIST
	stParentPath := '';
	stParentPath := CONCAT('//*/objLst/obj[@id=$'',CONCAT(stBacNetDeviceId,'$']'));	
	IF fcXMLAddNode(stParentPath,'p','id',TO_STRING(TO_INT(WagoTypesBACnet.eBACnetPropertyIdentifier.PROP_STRUCTURED_OBJECT_LIST)),'s','1',stXmlPath,FALSE) THEN	
		fcXMLAddStructuredViewToDevice := TRUE;
	END_IF;
		// Check if Node exist
		stParentPath := '';
		stParentPath := CONCAT(CONCAT(CONCAT(CONCAT('//*/objLst/obj[@id=$'',stBacNetDeviceId),'$']/p[@id=$''),TO_STRING(TO_INT(WagoTypesBACnet.eBACnetPropertyIdentifier.PROP_STRUCTURED_OBJECT_LIST))),'$']');	
		IF NOT fcXMLCheckNode(stParentPath,'n','t','192','v',stBacNetStructView,stXmlPath) THEN
			// Create Node 192 PROP_STRUCTURED_OBJECT_LIST
			stParentPath := '';
			stParentPath := CONCAT(CONCAT(CONCAT(CONCAT('//*/objLst/obj[@id=$'',stBacNetDeviceId),'$']/p[@id=$''),TO_STRING(TO_INT(WagoTypesBACnet.eBACnetPropertyIdentifier.PROP_STRUCTURED_OBJECT_LIST))),'$']');	
			IF fcXMLAddNode(stParentPath,'n','t','192','v',stBacNetStructView,stXmlPath,TRUE) THEN	
				fcXMLAddStructuredViewToDevice := TRUE;
			END_IF;
		END_IF;
		// Set Reboot Required
		IF fcXMLAddStructuredViewToDevice THEN
			GVL_BACNET.fbBacNetParameter.proRebootRequired := TRUE;
		END_IF;
END_IF;

END_FUNCTION

// 30 Program Organization Units/FBs/AT_FUNKTIONEN/AT_MESSWERTGEBER_STETIG/FB_AT_MESSWERTGEBER_STETIG
FUNCTION_BLOCK FB_AT_MESSWERTGEBER_STETIG EXTENDS FB_OBJ_ID_BASE
VAR_INPUT
	rValue				:	REAL;
	rLowLim				:	REAL;
	rHighLim			:	REAL;
	rMinPresValue		:	REAL;
	rMaxPresValue		:	REAL;
	enUnit				:	WagoTypesBACnet.eBACnetUnits;
END_VAR
VAR_OUTPUT
	(* Requests *)
	xHandPrio8	:	BOOL;
END_VAR
VAR
	(* BacNet Objects *)
	A_AI_1		:	WagoSysBACnet.FbAnalogInput_large(-1);					// Istwert
	B_EE_1		:	WagoSysBACnet.FbEventEnrollment_large(-1);              // Voralarm
	C_TL_1		:	WagoSysBACnet.FbTrendLog_large(-1);                     // Aufzeichnung Istwert

END_VAR
VAR CONSTANT
	usiAnzBacNetObj	:	USINT	:= 3;
END_VAR

(* Call Base FB*)
SUPER^();
(* Cyclic Action *)
IF xCreatet THEN
	(* DESCTIPTION FIX *)
	metCYCLIC_DESCRIPTION_FIX();
	(* Get Revision *)
	CASE GVL_BACNET.fbBacNetParameter.proKBOB_REV OF
		(* KBOB 2021 V2 *)
		enKBOB_REV.KBOB_REV2021_V2:
			metCYCLIC_KBOB_2021_V2();
		(* KBOB 2017 V1 *)
		enKBOB_REV.KBOB_REV2017_V1:
			metCYCLIC_KBOB_2017_V1();
		(* Default *)
		ELSE
			metCYCLIC_KBOB_2021_V2();
	END_CASE;	
END_IF;

METHOD metDELETE : BOOL
VAR_INPUT
END_VAR
VAR
	oStatus		:	WagoSysErrorBase.FbResult;
	usiErrors	:	USINT;
END_VAR
(* A_BO_1*)
IF A_AI_1.xIsCreated THEN
	A_AI_1.Delete(oStatus=>oStatus);
END_IF;	
(* B_EE_1 *)
IF B_EE_1.xIsCreated THEN
	B_EE_1.Delete(oStatus=>oStatus);	
END_IF;
(* C_TL_1 *)
IF C_TL_1.xIsCreated THEN
	IF GVL_BACNET.fbBacNetParameter.proDestroyBacNetOverrideXmlNode THEN
		fcXMLDeleteOverrideNode(fcBacNetIdToIdWitType(C_TL_1.IObjectIdentifier.diInstance,C_TL_1.IObjectIdentifier.eObjectType));
	END_IF;
	C_TL_1.Delete(oStatus=>oStatus);	
END_IF;
(* Delete Struct View *)
IF GVL_BACNET.fbBacNetParameter.proDestroyBacNetOverrideXmlNode THEN
	fcXMLDeleteOverrideNode(fcBacNetIdToIdWitType(TO_DINT(CONCAT(TO_STRING(OBJ_ID_BASE),'1')),WagoTypesBacNet.eBACnetObjectType.BACnet_structured_view));
	fcXMLDeleteStructuredViewFromDevice(fcBacNetIdToIdWitType(TO_DINT(CONCAT(TO_STRING(OBJ_ID_BASE),'1')),WagoTypesBacNet.eBACnetObjectType.BACnet_structured_view));
END_IF;
metDELETE :=	A_AI_1.xIsCreated OR
				C_TL_1.xIsCreated OR
				B_EE_1.xIsCreated ;
(* Reset Create Case *)
usiCreateCase := 1;
END_METHOD

(*FB_Exit muss explizit implementiert werden. Wenn es eine Implementierung gibt, dann wird 
die Methode aufgerufen, bevor die Steuerung den Code der Funktionsbaustein-Instanz entfernt
(impliziter Aufruf. Der Rückgabewert wird nicht ausgewertet.*)
METHOD FB_Exit : BOOL
VAR_INPUT
	(* TRUE: Die Exit-Methode wird aufgerufen, um die Instanz zu verlassen, die hinterher kopiert wird Online-Change).  *)
	bInCopyCode	: BOOL;
END_VAR
(* A_BO_1*)
IF A_AI_1.xIsCreated THEN
	A_AI_1.Delete();
END_IF;	
(* B_TL_1 *)
IF C_TL_1.xIsCreated THEN
	C_TL_1.Delete();	
END_IF;
(* C_EE_1 *)
IF B_EE_1.xIsCreated THEN
	B_EE_1.Delete();	
END_IF;
END_METHOD

METHOD metCREATE : BOOL;
VAR_INPUT
END_VAR
VAR
	usiErrors	:	USINT;
END_VAR
(* Get Revision *)
CASE GVL_BACNET.fbBacNetParameter.proKBOB_REV OF
	(* KBOB 2021 V2 *)
	enKBOB_REV.KBOB_REV2021_V2:
		usiErrors := usiErrors + TO_USINT(NOT metCREATE_KBOB_2021_V2());
	(* KBOB 2017 V1 *)
	enKBOB_REV.KBOB_REV2017_V1:
		usiErrors := usiErrors + TO_USINT(NOT metCREATE_KBOB_2017_V1());
	(* Default *)
	ELSE
		usiErrors := usiErrors + TO_USINT(NOT metCREATE_KBOB_2021_V2());
END_CASE;

(* OK = 0*)
xErrorCreate := TO_BOOL(usiErrors);
metCREATE := NOT TO_BOOL(usiErrors) AND usiCreateCase = usiAnzBacNetObj;
END_METHOD

METHOD metCreate_A_AI_1 : BOOL
(* A_AI_1*)
IF NOT A_AI_1.xIsCreated THEN
	(* Ziel						UTF8->ASCII						OBJ_NAME_BASE			BacNet Text		Textlistname									BacNet Funktion																	BacNet Textlist type												TextId		*)
	A_AI_1._sObjectName		:=	fcUtfToAscii(Standard.CONCAT(	OBJ_NAME_BASE		,	fcGetBcText(	GVL_BACNET.fbBacNetParameter.metGetTextListName(enTypeOfBacNetFunktionIn := enTypeOfBacNetFunktion.Type_MesswertgeberStetig,	enTypeOfBacNetTextListIn := enTypeOfBacNetTextList.ENDING		),	'A_AI_1')));
	A_AI_1._sDescription	:= 	fcUtfToAscii(Standard.CONCAT(	OBJ_NAME_DESCRIPTION,	fcGetBcText(	GVL_BACNET.fbBacNetParameter.metGetTextListName(enTypeOfBacNetFunktionIn := enTypeOfBacNetFunktion.Type_MesswertgeberStetig,	enTypeOfBacNetTextListIn := enTypeOfBacNetTextList.DESCRIPTION	),	'A_AI_1')));
	(* Create Id from Base Id and Object Nr (Last nummber of Name *)	
	A_AI_1.Create(diInstance := TO_DINT(Standard.CONCAT(TO_STRING(dwOBJ_ID_BASE),'1')));
	(* Check if Created *)
	IF A_AI_1.xIsCreated THEN
		(* Set Group *)
		A_AI_1.setPropertyGroup(WagoTypesBacNet.eBACnetPropertyIdentifier.PROP_PRESENT_VALUE						,WagoTypesBacNet.eBACnetPropertyUpdateGroup.GROUP_CYCLIC);
		A_AI_1.setPropertyGroup(WagoTypesBacNet.eBACnetPropertyIdentifier.PROP_PRIORITY_ARRAY						,WagoTypesBacNet.eBACnetPropertyUpdateGroup.GROUP_CYCLIC);
		A_AI_1.setPropertyGroup(WagoTypesBacNet.eBACnetPropertyIdentifier.PROP_ELAPSED_ACTIVE_TIME					,WagoTypesBacNet.eBACnetPropertyUpdateGroup.GROUP_CYCLIC);
		A_AI_1.setPropertyGroup(WagoTypesBacNet.eBACnetPropertyIdentifier.PROP_DESCRIPTION							,WagoTypesBacNet.eBACnetPropertyUpdateGroup.GROUP_CYCLIC);
		A_AI_1.setPropertyGroup(WagoTypesBacNet.eBACnetPropertyIdentifier.PROP_EVENT_MESSAGE_TEXTS_CONFIG			,WagoTypesBacNet.eBACnetPropertyUpdateGroup.GROUP_CYCLIC);
		(* Set Description to Overwrite retain*)
		A_AI_1.sDescription	:= A_AI_1._sDescription;
		(* Ziel												UTF8->ASCII		BacNet Text		Textlistname									BacNet Funktion																	BacNet Textlist type												TextId		*)
		A_AI_1.IEventMessageTextsConfig.sToOffNormal	:=	fcUtfToAscii(	fcGetBcText(	GVL_BACNET.fbBacNetParameter.metGetTextListName(enTypeOfBacNetFunktionIn := enTypeOfBacNetFunktion.Type_MesswertgeberStetig,	enTypeOfBacNetTextListIn := enTypeOfBacNetTextList.EVENTMESSAGE	),	'A_AI_1_ToOffNormal'	));		
		A_AI_1.IEventMessageTextsConfig.sToFault		:=	fcUtfToAscii(	fcGetBcText(	GVL_BACNET.fbBacNetParameter.metGetTextListName(enTypeOfBacNetFunktionIn := enTypeOfBacNetFunktion.Type_MesswertgeberStetig,	enTypeOfBacNetTextListIn := enTypeOfBacNetTextList.EVENTMESSAGE	),	'A_AI_1_ToFault'		));		
		A_AI_1.IEventMessageTextsConfig.sToNormal		:=	fcUtfToAscii(	fcGetBcText(	GVL_BACNET.fbBacNetParameter.metGetTextListName(enTypeOfBacNetFunktionIn := enTypeOfBacNetFunktion.Type_MesswertgeberStetig,	enTypeOfBacNetTextListIn := enTypeOfBacNetTextList.EVENTMESSAGE	),	'A_AI_1_ToNormal'		));		

		(* Ziel												Convert			BacNet Text		Textlistname									BacNet Funktion																	BacNet Textlist type												TextId		*)	
		A_AI_1.udiNotificationClass						:= 	TO_UDINT	(	fcGetBcText(	GVL_BACNET.fbBacNetParameter.metGetTextListName(enTypeOfBacNetFunktionIn := enTypeOfBacNetFunktion.Type_MesswertgeberStetig,	enTypeOfBacNetTextListIn := enTypeOfBacNetTextList.NC			),	'A_AI_1_NC'	));	
		A_AI_1.eNotifyType								:= 	WagoTypesBACnet.eBACnetNotifyType.NOTIFY_TYPE_EVENT;
		
	ELSE
		A_AI_1.Delete();
	END_IF;
	(* Get Status *)
	metCreate_A_AI_1 := A_AI_1.xIsCreated;	
END_IF;
END_METHOD

METHOD metCreate_C_TL_1 : BOOL
(* C_TL_1*)
IF NOT C_TL_1.xIsCreated THEN
	(* Ziel						UTF8->ASCII						OBJ_NAME_BASE			BacNet Text		Textlistname									BacNet Funktion																	BacNet Textlist type												TextId		*)
	C_TL_1._sObjectName		:=	fcUtfToAscii(Standard.CONCAT(	OBJ_NAME_BASE		,	fcGetBcText(	GVL_BACNET.fbBacNetParameter.metGetTextListName(enTypeOfBacNetFunktionIn := enTypeOfBacNetFunktion.Type_MesswertgeberStetig,	enTypeOfBacNetTextListIn := enTypeOfBacNetTextList.ENDING		),	'C_TL_1')));
	C_TL_1._sDescription	:= 	fcUtfToAscii(Standard.CONCAT(	OBJ_NAME_DESCRIPTION,	fcGetBcText(	GVL_BACNET.fbBacNetParameter.metGetTextListName(enTypeOfBacNetFunktionIn := enTypeOfBacNetFunktion.Type_MesswertgeberStetig,	enTypeOfBacNetTextListIn := enTypeOfBacNetTextList.DESCRIPTION	),	'C_TL_1')));
	(* Create Id from Base Id and Object Nr (Last nummber of Name *)	
	C_TL_1.Create(diInstance := TO_DINT(Standard.CONCAT(TO_STRING(dwOBJ_ID_BASE),'1')));
	(* Check if Created *)
	IF C_TL_1.xIsCreated THEN
		(* Set Group *)
		C_TL_1.setPropertyGroup(WagoTypesBacNet.eBACnetPropertyIdentifier.PROP_PRESENT_VALUE						,WagoTypesBacNet.eBACnetPropertyUpdateGroup.GROUP_CYCLIC);
		C_TL_1.setPropertyGroup(WagoTypesBacNet.eBACnetPropertyIdentifier.PROP_PRIORITY_ARRAY						,WagoTypesBacNet.eBACnetPropertyUpdateGroup.GROUP_CYCLIC);
		C_TL_1.setPropertyGroup(WagoTypesBacNet.eBACnetPropertyIdentifier.PROP_ELAPSED_ACTIVE_TIME					,WagoTypesBacNet.eBACnetPropertyUpdateGroup.GROUP_CYCLIC);
		C_TL_1.setPropertyGroup(WagoTypesBacNet.eBACnetPropertyIdentifier.PROP_DESCRIPTION							,WagoTypesBacNet.eBACnetPropertyUpdateGroup.GROUP_CYCLIC);
		C_TL_1.setPropertyGroup(WagoTypesBacNet.eBACnetPropertyIdentifier.PROP_EVENT_MESSAGE_TEXTS_CONFIG			,WagoTypesBacNet.eBACnetPropertyUpdateGroup.GROUP_CYCLIC);
		(* Crate Override *)
		fcXMLTrendLogOverride(C_TL_1,A_AI_1.IObjectIdentifier,WagoTypesBacNet.eBACnetPropertyIdentifier.PROP_PRESENT_VALUE);
		(* Set Description to Overwrite retain*)
		C_TL_1.sDescription	:= C_TL_1._sDescription;
		(* Ziel												UTF8->ASCII		BacNet Text		Textlistname									BacNet Funktion																	BacNet Textlist type												TextId		*)
		C_TL_1.IEventMessageTextsConfig.sToOffNormal	:=	fcUtfToAscii(	fcGetBcText(	GVL_BACNET.fbBacNetParameter.metGetTextListName(enTypeOfBacNetFunktionIn := enTypeOfBacNetFunktion.Type_MesswertgeberStetig,	enTypeOfBacNetTextListIn := enTypeOfBacNetTextList.EVENTMESSAGE	),	'C_TL_1_ToOffNormal'	));		
		C_TL_1.IEventMessageTextsConfig.sToFault		:=	fcUtfToAscii(	fcGetBcText(	GVL_BACNET.fbBacNetParameter.metGetTextListName(enTypeOfBacNetFunktionIn := enTypeOfBacNetFunktion.Type_MesswertgeberStetig,	enTypeOfBacNetTextListIn := enTypeOfBacNetTextList.EVENTMESSAGE	),	'C_TL_1_ToFault'		));		
		C_TL_1.IEventMessageTextsConfig.sToNormal		:=	fcUtfToAscii(	fcGetBcText(	GVL_BACNET.fbBacNetParameter.metGetTextListName(enTypeOfBacNetFunktionIn := enTypeOfBacNetFunktion.Type_MesswertgeberStetig,	enTypeOfBacNetTextListIn := enTypeOfBacNetTextList.EVENTMESSAGE	),	'C_TL_1_ToNormal'		));		
		(* Ziel												Convert			BacNet Text		Textlistname									BacNet Funktion																	BacNet Textlist type												TextId		*)	
		C_TL_1.udiNotificationClass						:= 	TO_UDINT	(	fcGetBcText(	GVL_BACNET.fbBacNetParameter.metGetTextListName(enTypeOfBacNetFunktionIn := enTypeOfBacNetFunktion.Type_MesswertgeberStetig,	enTypeOfBacNetTextListIn := enTypeOfBacNetTextList.NC			),	'C_TL_1_NC'	));	
		C_TL_1.eNotifyType								:= 	WagoTypesBACnet.eBACnetNotifyType.NOTIFY_TYPE_EVENT;
	
		(* Logging Type *)
		C_TL_1.eLoggingType								:= WagoTypesBACnet.eBACnetLoggingType.LOGGING_TYPE_POLLED;
	
		(* Activate Logging *)
		C_TL_1.xEnable	:= TRUE;
		
	ELSE
		C_TL_1.Delete();
	END_IF;
	(* Get Status *)
	metCreate_C_TL_1 := C_TL_1.xIsCreated;	
END_IF;
END_METHOD

METHOD metCreate_B_EE_1 : BOOL
(* B_EE_1*)
IF NOT B_EE_1.xIsCreated THEN
	(* Ziel						UTF8->ASCII						OBJ_NAME_BASE			BacNet Text		Textlistname									BacNet Funktion																	BacNet Textlist type												TextId		*)
	B_EE_1._sObjectName		:=	fcUtfToAscii(Standard.CONCAT(	OBJ_NAME_BASE		,	fcGetBcText(	GVL_BACNET.fbBacNetParameter.metGetTextListName(enTypeOfBacNetFunktionIn := enTypeOfBacNetFunktion.Type_MesswertgeberStetig,	enTypeOfBacNetTextListIn := enTypeOfBacNetTextList.ENDING		),	'B_EE_1')));
	B_EE_1._sDescription	:= 	fcUtfToAscii(Standard.CONCAT(	OBJ_NAME_DESCRIPTION,	fcGetBcText(	GVL_BACNET.fbBacNetParameter.metGetTextListName(enTypeOfBacNetFunktionIn := enTypeOfBacNetFunktion.Type_MesswertgeberStetig,	enTypeOfBacNetTextListIn := enTypeOfBacNetTextList.DESCRIPTION	),	'B_EE_1')));
	(* Create Id from Base Id and Object Nr (Last nummber of Name *)	
	B_EE_1.Create(diInstance := TO_DINT(Standard.CONCAT(TO_STRING(dwOBJ_ID_BASE),'1')));
	(* Check if Created *)
	IF B_EE_1.xIsCreated THEN
		(* Set Group *)
		B_EE_1.setPropertyGroup(WagoTypesBacNet.eBACnetPropertyIdentifier.PROP_PRESENT_VALUE						,WagoTypesBacNet.eBACnetPropertyUpdateGroup.GROUP_CYCLIC);
		B_EE_1.setPropertyGroup(WagoTypesBacNet.eBACnetPropertyIdentifier.PROP_PRIORITY_ARRAY						,WagoTypesBacNet.eBACnetPropertyUpdateGroup.GROUP_CYCLIC);
		B_EE_1.setPropertyGroup(WagoTypesBacNet.eBACnetPropertyIdentifier.PROP_ELAPSED_ACTIVE_TIME					,WagoTypesBacNet.eBACnetPropertyUpdateGroup.GROUP_CYCLIC);
		B_EE_1.setPropertyGroup(WagoTypesBacNet.eBACnetPropertyIdentifier.PROP_DESCRIPTION							,WagoTypesBacNet.eBACnetPropertyUpdateGroup.GROUP_CYCLIC);
		B_EE_1.setPropertyGroup(WagoTypesBacNet.eBACnetPropertyIdentifier.PROP_EVENT_MESSAGE_TEXTS_CONFIG			,WagoTypesBacNet.eBACnetPropertyUpdateGroup.GROUP_CYCLIC);
		(* Set Description to Overwrite retain*)
		B_EE_1.sDescription	:= B_EE_1._sDescription;
		(* Ziel												UTF8->ASCII		BacNet Text		Textlistname									BacNet Funktion																	BacNet Textlist type												TextId		*)
		B_EE_1.IEventMessageTextsConfig.sToOffNormal	:=	fcUtfToAscii(	fcGetBcText(	GVL_BACNET.fbBacNetParameter.metGetTextListName(enTypeOfBacNetFunktionIn := enTypeOfBacNetFunktion.Type_MesswertgeberStetig,	enTypeOfBacNetTextListIn := enTypeOfBacNetTextList.EVENTMESSAGE	),	'B_EE_1_ToOffNormal'	));		
		B_EE_1.IEventMessageTextsConfig.sToFault		:=	fcUtfToAscii(	fcGetBcText(	GVL_BACNET.fbBacNetParameter.metGetTextListName(enTypeOfBacNetFunktionIn := enTypeOfBacNetFunktion.Type_MesswertgeberStetig,	enTypeOfBacNetTextListIn := enTypeOfBacNetTextList.EVENTMESSAGE	),	'B_EE_1_ToFault'		));		
		B_EE_1.IEventMessageTextsConfig.sToNormal		:=	fcUtfToAscii(	fcGetBcText(	GVL_BACNET.fbBacNetParameter.metGetTextListName(enTypeOfBacNetFunktionIn := enTypeOfBacNetFunktion.Type_MesswertgeberStetig,	enTypeOfBacNetTextListIn := enTypeOfBacNetTextList.EVENTMESSAGE	),	'B_EE_1_ToNormal'		));		

		(* Ziel												Convert			BacNet Text		Textlistname									BacNet Funktion																	BacNet Textlist type												TextId		*)	
		B_EE_1.udiNotificationClass						:= 	TO_UDINT	(	fcGetBcText(	GVL_BACNET.fbBacNetParameter.metGetTextListName(enTypeOfBacNetFunktionIn := enTypeOfBacNetFunktion.Type_MesswertgeberStetig,	enTypeOfBacNetTextListIn := enTypeOfBacNetTextList.NC			),	'B_EE_1_NC'	));	
		B_EE_1.eNotifyType								:= 	WagoTypesBACnet.eBACnetNotifyType.NOTIFY_TYPE_ALARM;
		
	ELSE
		B_EE_1.Delete();
	END_IF;
	(* Get Status *)
	metCreate_B_EE_1 := B_EE_1.xIsCreated;	
END_IF;
END_METHOD

METHOD metCREATE_KBOB_2017_V1 : BOOL;
VAR_INPUT
END_VAR
VAR
	oStatus		:	WagoSysErrorBase.FbResult;
	usiErrors	:	USINT;
END_VAR
(* Resett *)
usiErrors := 0;	

(* Create Objeccts *)
CASE usiCreateCase OF
	1:	
		usiErrors := usiErrors + TO_USINT(NOT metCreate_A_AI_1());
	2:
		usiErrors := usiErrors + TO_USINT(NOT metCreate_B_EE_1());
	3:	
		usiErrors := usiErrors + TO_USINT(NOT metCreate_C_TL_1());
	0: 
		usiCreateCase := 1;
ELSE
	usiCreateCase := 0;
END_CASE;

(* STRUCT VIEW *)
metCREATE_STRUCTVIEW_KBOB_2017_V1();

(* OK = 0*)
metCREATE_KBOB_2017_V1 := NOT TO_BOOL(usiErrors);
END_METHOD

METHOD metCREATE_STRUCTVIEW_KBOB_2017_V1 : BOOL
VAR_INPUT
END_VAR
CASE usiCreateCase OF
	1:	
		fcXMLStructuredView(THIS^,A_AI_1.IObjectIdentifier);
	2:
		fcXMLStructuredView(THIS^,B_EE_1.IObjectIdentifier);
	3:
		fcXMLStructuredView(THIS^,C_TL_1.IObjectIdentifier);
		fcXMLAddStructuredViewToDevice(THIS^);
	0: 
		usiCreateCase := 1;
ELSE
	usiCreateCase := 0;
END_CASE
END_METHOD

METHOD metCREATE_KBOB_2021_V2 : BOOL;
VAR_INPUT
END_VAR
VAR
	oStatus		:	WagoSysErrorBase.FbResult;
	usiErrors	:	USINT;
END_VAR
(* Resett *)
usiErrors := 0;	

(* Create Objeccts *)
CASE usiCreateCase OF
	1:	
		usiErrors := usiErrors + TO_USINT(NOT metCreate_A_AI_1());
	2:
		usiErrors := usiErrors + TO_USINT(NOT metCreate_B_EE_1());
	3:	
		usiErrors := usiErrors + TO_USINT(NOT metCreate_C_TL_1());
	0: 
		usiCreateCase := 1;
ELSE
	usiCreateCase := 0;
END_CASE;

(* STRUCT VIEW *)
metCREATE_STRUCTVIEW_KBOB_2021_V2();

(* OK = 0*)
metCREATE_KBOB_2021_V2 := NOT TO_BOOL(usiErrors);
END_METHOD

METHOD metCREATE_STRUCTVIEW_KBOB_2021_V2 : BOOL
VAR_INPUT
END_VAR
CASE usiCreateCase OF
	1:	
		fcXMLStructuredView(THIS^,A_AI_1.IObjectIdentifier);
	2:
		fcXMLStructuredView(THIS^,B_EE_1.IObjectIdentifier);
	3:
		fcXMLStructuredView(THIS^,C_TL_1.IObjectIdentifier);
		fcXMLAddStructuredViewToDevice(THIS^);
	0: 
		usiCreateCase := 1;
ELSE
	usiCreateCase := 0;
END_CASE
END_METHOD

METHOD metCYCLIC_KBOB_2017_V1
VAR_INPUT
END_VAR
(* A_BO_1 *)
IF A_AI_1.rIN <> rValue THEN
	A_AI_1.rIN := rValue;				
END_IF;
IF A_AI_1.rLowLimit <> rLowLim THEN
	A_AI_1.rLowLimit := rLowLim;	
END_IF;
IF A_AI_1.rHighLimit <> rHighLim THEN
	A_AI_1.rHighLimit := rHighLim;	
END_IF;
IF A_AI_1._rMinPresValue <> rMinPresValue THEN
	A_AI_1._rMinPresValue := rMinPresValue;	
END_IF;
IF A_AI_1._rMaxPresValue <> rMaxPresValue THEN
	A_AI_1._rMaxPresValue := rMaxPresValue;	
END_IF;
END_METHOD

METHOD metCYCLIC_KBOB_2021_V2
VAR_INPUT
END_VAR
(* A_BO_1 *)
IF A_AI_1.rIN <> rValue THEN
	A_AI_1.rIN := rValue;				
END_IF;
IF A_AI_1.rLowLimit <> rLowLim THEN
	A_AI_1.rLowLimit := rLowLim;	
END_IF;
IF A_AI_1.rHighLimit <> rHighLim THEN
	A_AI_1.rHighLimit := rHighLim;	
END_IF;
IF A_AI_1._rMinPresValue <> rMinPresValue THEN
	A_AI_1._rMinPresValue := rMinPresValue;	
END_IF;
IF A_AI_1._rMaxPresValue <> rMaxPresValue THEN
	A_AI_1._rMaxPresValue := rMaxPresValue;	
END_IF;
END_METHOD

METHOD metCYCLIC_DESCRIPTION_FIX
VAR_INPUT
END_VAR
(* A_AI_1 *)
IF A_AI_1.xIsCreated THEN
	IF A_AI_1.sDescription <> A_AI_1._sDescription THEN
		A_AI_1.sDescription := A_AI_1._sDescription;
	END_IF;
END_IF;

(* B_EE_1 *)
IF B_EE_1.xIsCreated THEN
	IF B_EE_1.sDescription <> B_EE_1._sDescription THEN
		B_EE_1.sDescription := B_EE_1._sDescription;
	END_IF;
END_IF;

(* C_TL_1 *)
IF C_TL_1.xIsCreated THEN
	IF C_TL_1.sDescription <> C_TL_1._sDescription THEN
		C_TL_1.sDescription := C_TL_1._sDescription;
	END_IF;
END_IF;
END_METHOD

END_FUNCTION_BLOCK

// 30 Program Organization Units/FCs/XMLFcs/XMLBase/fcXMLUpdateNode
FUNCTION fcXMLUpdateNode : BOOL
VAR_INPUT
	stParentPath		:	STRING(80);	// Start with '//*/
	stNodeName			:	STRING(15);
	stXmlFilePathName	:	STRING(80);
END_VAR
VAR
	stCommand			:	STRING(255);
	stResult			:	STRING(255);
	RTS_IEC_RESULT		:	SysTypes.RTS_IEC_RESULT;
END_VAR

stCommand := 	'';
stCommand := 	Standard.CONCAT(
				Standard.CONCAT(
				Standard.CONCAT(
				Standard.CONCAT(
				Standard.CONCAT(
								'xmlstarlet ed -L --update "',	
								stParentPath),
								'" -t elem -n "'),
								stNodeName),
								'" '),
								stXmlFilePathName);
SysProcess_Implementation.SysProcessExecuteCommand(stCommand,RTS_IEC_RESULT);

END_FUNCTION

